// TwinCAT 3 PLC project Depal2
// libraries:
//   Tc2_Standard, * (Beckhoff Automation GmbH)
//   Tc2_System, * (Beckhoff Automation GmbH)
//   Tc3_Module, * (Beckhoff Automation GmbH)
// project tree:
//   Global Variables/ Global_Variables.TcGVL, Global_Variables_HMI.TcGVL, Global_Variables_sBool.TcGVL, Variable_Configuration.TcGVL
//   POUs/Function Blocks/ TOGGLE.TcPOU
//   POUs/ IOLink.TcPOU, MAIN.TcPOU, Messages.TcPOU, Tiersheet_Car.TcPOU
//   / Standard.TcTTO
// real-time tasks:
//   TASK Standard: cycle T#10ms, priority 20, ADS port 350
// I/O:
//   DEVICE Depal 2 I/O, AmsNetId 5.155.243.167.3.1
//     Term 1 (EK1200) [EK1200-5000 EtherCAT Power supply (2A E-Bus)]
//       Term 2 (EK1122) [EK1122 2 port EtherCAT junction]
//         IO-Link1 (ifm IO-Link Master AL1332) [ifm IO-Link Master AL1332]
//           modules: Module 1 (IOL_In_8Byte), Module 2 (IOL_In_8Byte), Module 3 (IOL_In_8Byte), Module 4 (IOL_In_8Byte), Module 5 (IOL_In_8Byte), Module 6 (IOL_In_8Byte), Module 7 (IOL_In_8Byte), Module 8 (IOL_In_8Byte)
//         IO-Link2 (ifm IO-Link Master AL1332) [ifm IO-Link Master AL1332]
//           modules: Module 1 (IOL_In_8Byte), Module 2 (IOL_In_8Byte), Module 3 (IOL_In_8Byte), Module 4 (IOL_In_8Byte), Module 5 (IOL_In_8Byte), Module 6 (IOL_In_8Byte), Module 7 (IOL_In_8Byte), Module 8 (IOL_In_8Byte)
//         IO-Link3 (ifm IO-Link Master AL1332) [ifm IO-Link Master AL1332]
//           modules: Module 1 (IOL_In_8Byte), Module 2 (IOL_In_8Byte), Module 3 (IOL_In_8Byte), Module 4 (IOL_In_8Byte), Module 5 (IOL_In_8Byte), Module 6 (IOL_In_8Byte), Module 7 (IOL_In_8Byte), Module 8 (IOL_In_8Byte)
//         IO-Link4 (ifm IO-Link Master AL1332) [ifm IO-Link Master AL1332]
//           modules: Module 1 (IOL_In_8Byte), Module 2 (IOL_In_8Byte), Module 3 (IOL_In_8Byte), Module 4 (IOL_In_8Byte), Module 5 (IOL_In_8Byte), Module 6 (IOL_In_8Byte), Module 7 (IOL_In_8Byte), Module 8 (IOL_In_8Byte)
//         IO-Link5 (ifm IO-Link Master AL1332) [ifm IO-Link Master AL1332]
//           modules: Module 1 (IOL_In_8Byte), Module 2 (Digital_IN), Module 3 (Digital_IN), Module 4 (IOL_In_8Byte), Module 5 (IOL_In_8Byte), Module 6 (IOL_In_8Byte), Module 7 (IOL_In_8Byte), Module 8 (IOL_In_8Byte)
//       Box 4 (BK1250)
// variable links:
//   Depal2/Depal2 Instance <-> Depal 2 I/O/Term 1 (EK1200)/Box 4 (BK1250)
//     Standard Inputs/.i453 <-> Term 7 (KL1114)/Channel 4/Input
//     Standard Inputs/.iCarriage_VAC <-> Term 2 (KL1114)/Channel 3/Input
//     Standard Inputs/.iCarriage_Vfd <-> Term 5 (KL1114)/Channel 3/Input
//     Standard Inputs/.iChain_Hoist_VAC <-> Term 2 (KL1114)/Channel 2/Input
//     Standard Inputs/.iChain_Hoist_Vfd <-> Term 5 (KL1114)/Channel 2/Input
//     Standard Inputs/.iChamber_Chain_VAC <-> Term 2 (KL1114)/Channel 4/Input
//     Standard Inputs/.iChamber_Chain_Vfd <-> Term 5 (KL1114)/Channel 4/Input
//     Standard Inputs/.iDM2_EmergencyStop <-> Term 8 (KL9260)/Channel 1/Power
//     Standard Inputs/.iDM2_Fuse <-> Term 8 (KL9260)/Channel 1/ShortCircuit
//     Standard Inputs/.iDischarge1_VAC <-> Term 4 (KL1114)/Channel 1/Input
//     Standard Inputs/.iDischarge2_VAC <-> Term 4 (KL1114)/Channel 2/Input
//     Standard Inputs/.iDischarge3_VAC <-> Term 4 (KL1114)/Channel 3/Input
//     Standard Inputs/.iDischarge1_Vfd <-> Term 7 (KL1114)/Channel 1/Input
//     Standard Inputs/.iDischarge2_Vfd <-> Term 7 (KL1114)/Channel 2/Input
//     Standard Inputs/.iDischarge3_Vfd <-> Term 7 (KL1114)/Channel 3/Input
//     Standard Inputs/.iPallet_Discharge_VAC <-> Term 3 (KL1114)/Channel 1/Input
//     Standard Inputs/.iPallet_Discharge_Vfd <-> Term 6 (KL1114)/Channel 1/Input
//     Standard Inputs/.iPallet_Infeed1_VAC <-> Term 3 (KL1114)/Channel 2/Input
//     Standard Inputs/.iPallet_Infeed2_VAC <-> Term 3 (KL1114)/Channel 3/Input
//     Standard Inputs/.iPallet_Infeed1_Vfd <-> Term 6 (KL1114)/Channel 2/Input
//     Standard Inputs/.iPallet_Infeed2_Vfd <-> Term 6 (KL1114)/Channel 3/Input
//     Standard Inputs/.iProductHeight_SweepPos <-> Term 4 (KL1114)/Channel 4/Input
//     Standard Inputs/.iTable_Top_VAC <-> Term 2 (KL1114)/Channel 1/Input
//     Standard Inputs/.iTable_Top_Vfd <-> Term 5 (KL1114)/Channel 1/Input
//     Standard Inputs/.iTierSheet_Car_VAC <-> Term 3 (KL1114)/Channel 4/Input
//     Standard Inputs/.iTierSheet_Car_Vfd <-> Term 6 (KL1114)/Channel 4/Input
//     Standard Outputs/.oBrake_Carriage <-> Term 30 (KL2612)/Channel 2/Output
//     Standard Outputs/.oBrake_Hoist <-> Term 30 (KL2612)/Channel 1/Output
//     Standard Outputs/.oCarriage_Forward <-> Term 25 (KL2612)/Channel 1/Output
//     Standard Outputs/.oCarriage_Reverse <-> Term 25 (KL2612)/Channel 2/Output
//     Standard Outputs/.oCarriage_Slow <-> Term 21 (KL2612)/Channel 2/Output
//     Standard Outputs/.oChainHoist_Down <-> Term 24 (KL2612)/Channel 2/Output
//     Standard Outputs/.oChainHoist_Up <-> Term 24 (KL2612)/Channel 1/Output
//     Standard Outputs/.oChainHoist_Up_Slow <-> Term 32 (KL2612)/Channel 1/Output
//     Standard Outputs/.oChainberChainRev <-> Term 32 (KL2612)/Channel 2/Output
//     Standard Outputs/.oDischarge1_Run <-> Term 28 (KL2612)/Channel 2/Output
//     Standard Outputs/.oDischarge2_Run <-> Term 29 (KL2612)/Channel 1/Output
//     Standard Outputs/.oElevator_Infeed <-> Term 26 (KL2612)/Channel 1/Output
//     Standard Outputs/.oHoistDoors_Close <-> Term 13 (KL2612)/Channel 2/Output
//     Standard Outputs/.oHoistDoors_Open <-> Term 13 (KL2612)/Channel 1/Output
//     Standard Outputs/.oHoist_Shrouds_Close <-> Term 12 (KL2612)/Channel 1/Output
//     Standard Outputs/.oHoist_Shrouds_Open <-> Term 12 (KL2612)/Channel 2/Output
//     Standard Outputs/.oIndicator_Green <-> Term 22 (KL2612)/Channel 1/Output
//     Standard Outputs/.oIndicator_Red <-> Term 23 (KL2612)/Channel 1/Output
//     Standard Outputs/.oIndicator_Yellow <-> Term 22 (KL2612)/Channel 2/Output
//     Standard Outputs/.oInfeed1Rev <-> Term 29 (KL2612)/Channel 2/Output
//     Standard Outputs/.oInfeed2Rev <-> Term 33 (KL2612)/Channel 1/Output
//     Standard Outputs/.oLayer_Capture <-> Term 14 (KL2612)/Channel 1/Output
//     Standard Outputs/.oLayer_Release <-> Term 14 (KL2612)/Channel 2/Output
//     Standard Outputs/.oPalletDischarge_Run <-> Term 26 (KL2612)/Channel 2/Output
//     Standard Outputs/.oPalletInfeed1_Run <-> Term 27 (KL2612)/Channel 1/Output
//     Standard Outputs/.oPalletInfeed2_Run <-> Term 27 (KL2612)/Channel 2/Output
//     Standard Outputs/.oSweepGate_Close <-> Term 9 (KL2612)/Channel 2/Output
//     Standard Outputs/.oSweepGate_Open <-> Term 9 (KL2612)/Channel 1/Output
//     Standard Outputs/.oSweepgate_Engage <-> Term 15 (KL2612)/Channel 1/Output
//     Standard Outputs/.oSweepgate_Release <-> Term 15 (KL2612)/Channel 2/Output
//     Standard Outputs/.oTableTop_Run <-> Term 23 (KL2612)/Channel 2/Output
//     Standard Outputs/.oTierSheetGripper_Engage <-> Term 16 (KL2612)/Channel 1/Output
//     Standard Outputs/.oTierSheetGripper_Release <-> Term 16 (KL2612)/Channel 2/Output
//     Standard Outputs/.oTierSheet_Bin_Close <-> Term 17 (KL2612)/Channel 2/Output
//     Standard Outputs/.oTierSheet_Bin_Open <-> Term 17 (KL2612)/Channel 1/Output
//     Standard Outputs/.oTierSheet_Car_Brake <-> Term 28 (KL2612)/Channel 1/Output
//     Standard Outputs/.oTierSheet_Car_Fwd <-> Term 31 (KL2612)/Channel 1/Output
//     Standard Outputs/.oTierSheet_Car_Rev <-> Term 31 (KL2612)/Channel 2/Output
//     Standard Outputs/.oTiersheetRemover_Down <-> Term 10 (KL2612)/Channel 2/Output
//     Standard Outputs/.oTiersheetRemover_Up <-> Term 10 (KL2612)/Channel 1/Output
//     Standard Outputs/.oTopFrame_Bin_Close <-> Term 18 (KL2612)/Channel 2/Output
//     Standard Outputs/.oTopFrame_Bin_Open <-> Term 18 (KL2612)/Channel 1/Output
//     Standard Outputs/.oTopFrame_Remover_Clamps_Engage <-> Term 20 (KL2612)/Channel 1/Output
//     Standard Outputs/.oTopFrame_Remover_Clamps_Release <-> Term 20 (KL2612)/Channel 2/Output
//     Standard Outputs/.oTopFrame_Remover_Lock <-> Term 19 (KL2612)/Channel 1/Output
//     Standard Outputs/.oTopFrame_Remover_Unlock <-> Term 19 (KL2612)/Channel 2/Output
//     Standard Outputs/.oTopFrame_Seize <-> Term 11 (KL2612)/Channel 2/Output
//     Standard Outputs/.oTrolleySlowdown <-> Term 33 (KL2612)/Channel 2/Output
//     Standard Outputs/.oVacuum_Engage <-> Term 21 (KL2612)/Channel 1/Output
//     Standard Outputs/.oVacuum_Solenoid <-> Term 11 (KL2612)/Channel 1/Output
//   Depal2/Depal2 Instance <-> Depal 2 I/O/Term 1 (EK1200)/Term 2 (EK1122)/IO-Link1 (ifm IO-Link Master AL1332)
//     Standard Inputs/.i1X01_HoistDoors_Closed <-> Module 1 (IOL_In_8Byte)/TxPDO/input byte 0
//     Standard Inputs/.i1X02_HoistLiftDown_Slowdown <-> Module 2 (IOL_In_8Byte)/TxPDO/input byte 0
//     Standard Inputs/.i1X03_HoistLift_Down <-> Module 3 (IOL_In_8Byte)/TxPDO/input byte 0
//     Standard Inputs/.i1X04_Hoist_Discharge_Jam <-> Module 4 (IOL_In_8Byte)/TxPDO/input byte 0
//     Standard Inputs/.i1X05_Infeed1_Pallet <-> Module 5 (IOL_In_8Byte)/TxPDO/input byte 0
//     Standard Inputs/.i1X06_Infeed2_Pallet <-> Module 6 (IOL_In_8Byte)/TxPDO/input byte 0
//     Standard Inputs/.i1X07_Pallet_in_Hoist <-> Module 7 (IOL_In_8Byte)/TxPDO/input byte 0
//     Standard Inputs/.i1X08_1114 <-> Module 8 (IOL_In_8Byte)/TxPDO/input byte 0
//   Depal2/Depal2 Instance <-> Depal 2 I/O/Term 1 (EK1200)/Term 2 (EK1122)/IO-Link2 (ifm IO-Link Master AL1332)
//     Standard Inputs/.i2X01 <-> Module 1 (IOL_In_8Byte)/TxPDO/input byte 0
//     Standard Inputs/.i2X02_HoistLift_Up <-> Module 2 (IOL_In_8Byte)/TxPDO/input byte 0
//     Standard Inputs/.i2X03_HoistLift_LastTier <-> Module 3 (IOL_In_8Byte)/TxPDO/input byte 0
//     Standard Inputs/.i2X04_Top_Frame_Monitor <-> Module 4 (IOL_In_8Byte)/TxPDO/input byte 0
//     Standard Inputs/.i2X05_DunnageBin_Full <-> Module 5 (IOL_In_8Byte)/TxPDO/input byte 0
//     Standard Inputs/.i2X06_TableTop_Accumulation <-> Module 6 (IOL_In_8Byte)/TxPDO/input byte 0
//     Standard Inputs/.i2X07_SingleFiler_Accumulation <-> Module 7 (IOL_In_8Byte)/TxPDO/input byte 0
//     Standard Inputs/.i2X08_CanTrack_Accumulation <-> Module 8 (IOL_In_8Byte)/TxPDO/input byte 0
//   Depal2/Depal2 Instance <-> Depal 2 I/O/Term 1 (EK1200)/Term 2 (EK1122)/IO-Link3 (ifm IO-Link Master AL1332)
//     Standard Inputs/.i3X01_SweepGateDoor_Open <-> Module 1 (IOL_In_8Byte)/TxPDO/input byte 0
//     Standard Inputs/.i3X02_CarriageRetract_Slowdown <-> Module 2 (IOL_In_8Byte)/TxPDO/input byte 0
//     Standard Inputs/.i3X03_Carriage_Retracted <-> Module 3 (IOL_In_8Byte)/TxPDO/input byte 0
//     Standard Inputs/.i3X04_Carriage_Extended <-> Module 4 (IOL_In_8Byte)/TxPDO/input byte 0
//     Standard Inputs/.i3X05_CarriageExtend_Slowdown <-> Module 5 (IOL_In_8Byte)/TxPDO/input byte 0
//     Standard Inputs/.i3X06_Layer_Capture_Monitor <-> Module 6 (IOL_In_8Byte)/TxPDO/input byte 0
//     Standard Inputs/.i3X07_Vacuum_On <-> Module 7 (IOL_In_8Byte)/TxPDO/input byte 0
//     Standard Inputs/.i3X08_ <-> Module 8 (IOL_In_8Byte)/TxPDO/input byte 0
//   Depal2/Depal2 Instance <-> Depal 2 I/O/Term 1 (EK1200)/Term 2 (EK1122)/IO-Link4 (ifm IO-Link Master AL1332)
//     Standard Inputs/.i4X01_Trolley_at_Hoist <-> Module 1 (IOL_In_8Byte)/TxPDO/input byte 0
//     Standard Inputs/.i4X02_Trolley_at_Hoist_Slowdown <-> Module 2 (IOL_In_8Byte)/TxPDO/input byte 0
//     Standard Inputs/.i4X03_Trolley_at_TierSheet_Bin_Slowdown <-> Module 3 (IOL_In_8Byte)/TxPDO/input byte 0
//     Standard Inputs/.i4X04_Trolley_at_TierSheetBin <-> Module 4 (IOL_In_8Byte)/TxPDO/input byte 0
//     Standard Inputs/.i4X05_Trolley_at_TopframeBin_Slowdown <-> Module 5 (IOL_In_8Byte)/TxPDO/input byte 0
//     Standard Inputs/.i4X06_Trolley_at_TopframeBin <-> Module 6 (IOL_In_8Byte)/TxPDO/input byte 0
//     Standard Inputs/.i4X07_TierSheetBin_Full <-> Module 7 (IOL_In_8Byte)/TxPDO/input byte 0
//     Standard Inputs/.i4X08_TopframeBin_Full <-> Module 8 (IOL_In_8Byte)/TxPDO/input byte 0
//   Depal2/Depal2 Instance <-> Depal 2 I/O/Term 1 (EK1200)/Term 2 (EK1122)/IO-Link5 (ifm IO-Link Master AL1332)
//     Standard Inputs/.i5X01_TierSheet_Vacuum_Monitor <-> Module 1 (IOL_In_8Byte)/TxPDO/input byte 0
//     Standard Inputs/.i5X02_TierSheet_Remover_Down <-> Module 2 (Digital_IN)/TxPDO/input byte 0
//     Standard Inputs/.i5X03_TiersheetRemoverUp <-> Module 3 (Digital_IN)/TxPDO/input byte 0
//     Standard Inputs/.i5X04_ <-> Module 4 (IOL_In_8Byte)/TxPDO/input byte 0
//     Standard Inputs/.i5X08_ <-> Module 8 (IOL_In_8Byte)/TxPDO/input byte 0
//     Standard Inputs/.i5X05_Topframe_Remover_Up <-> Module 5 (IOL_In_8Byte)/TxPDO/input byte 0
//     Standard Inputs/.i5X06_Topframe_On_BoardA <-> Module 6 (IOL_In_8Byte)/TxPDO/input byte 0
//     Standard Inputs/.i5X07_Topframe_On_BoardB <-> Module 7 (IOL_In_8Byte)/TxPDO/input byte 0

CONFIGURATION Depal2
    RESOURCE PLC ON TwinCAT3
        TASK Standard(INTERVAL := T#10ms, PRIORITY := 20);
        PROGRAM MAIN WITH Standard : MAIN;
    END_RESOURCE
END_CONFIGURATION

// ---- Global Variables/Global_Variables.TcGVL
{attribute 'Tc2GvlVarNames'}
VAR_GLOBAL
(***********************IO-LINK  INPUT************************************)
(**IO-Link1 AL1332**)
	i1X01_HoistDoors_Closed AT %I*:USINT;
	i1X02_HoistLiftDown_Slowdown AT %I*:USINT;
	i1X03_HoistLift_Down AT %I*:USINT;
	i1X04_Hoist_Discharge_Jam AT %I*:USINT;
	i1X05_Infeed1_Pallet AT %I*:USINT;
	i1X06_Infeed2_Pallet  AT %I*:USINT;
	i1X07_Pallet_in_Hoist AT %I*:USINT;
	i1X08_1114 AT %I*:USINT;

(**IO-Link2 AL1332**)
	i2X01 AT %I*:USINT;
	i2X02_HoistLift_Up AT %I*:USINT;
	i2X03_HoistLift_LastTier  AT %I*:USINT;
	i2X04_Top_Frame_Monitor AT %I*:USINT;
	i2X05_DunnageBin_Full AT %I*:USINT;
	i2X06_TableTop_Accumulation  AT %I*:USINT;
	i2X07_SingleFiler_Accumulation  AT %I*:USINT;
	i2X08_CanTrack_Accumulation  AT %I*:USINT;

(**IO-Link3 AL1332**)
	i3X01_SweepGateDoor_Open AT %I*:USINT;
	i3X02_CarriageRetract_Slowdown AT %I*:USINT;
	i3X03_Carriage_Retracted AT %I*:USINT;
	i3X04_Carriage_Extended AT %I*:USINT;
	i3X05_CarriageExtend_Slowdown AT %I*:USINT;
	i3X06_Layer_Capture_Monitor AT %I*:USINT;
	i3X07_Vacuum_On AT %I*:USINT;
	i3X08_ AT %I*:USINT;

(**IO-Link4 AL1332**)
	i4X01_Trolley_at_Hoist AT %I*:USINT;
	i4X02_Trolley_at_Hoist_Slowdown AT %I*:USINT;
	i4X03_Trolley_at_TierSheet_Bin_Slowdown AT %I*:USINT;
	i4X04_Trolley_at_TierSheetBin AT %I*:USINT;
	i4X05_Trolley_at_TopframeBin_Slowdown AT %I*:USINT;
	i4X06_Trolley_at_TopframeBin AT %I*:USINT;
	i4X07_TierSheetBin_Full AT %I*:USINT;
	i4X08_TopframeBin_Full AT %I*:USINT;

(**IO-Link5 AL1332**)
	i5X01_TierSheet_Vacuum_Monitor AT %I*:USINT;
	i5X02_TierSheet_Remover_Down AT %I*:USINT;
	i5X03_TiersheetRemoverUp AT %I*:USINT;
	i5X04_ AT %I*:USINT;
	i5X05_Topframe_Remover_Up AT %I*:USINT;
	i5X06_Topframe_On_BoardA AT %I*:USINT;
	i5X07_Topframe_On_BoardB AT %I*:USINT;
	i5X08_ AT %I*:USINT;

(**Slot 2 KL-1114*)(*VAC Disconnect*)
	iTable_Top_VAC AT %I*:BOOL;
	iChain_Hoist_VAC AT %I*:BOOL;
	iCarriage_VAC AT %I*:BOOL;
	iChamber_Chain_VAC AT %I*:BOOL;

(**Slot 3 KL1114*)(*VAC Disconnect*)
	iPallet_Discharge_VAC AT %I*:BOOL;
	iPallet_Infeed1_VAC AT %I*:BOOL;
	iPallet_Infeed2_VAC AT %I*:BOOL;
	iTierSheet_Car_VAC AT %I*:BOOL;

(**Slot 4 KL1114*)(*VAC Disconnect*)
	iDischarge1_VAC AT %I*:BOOL;
	iDischarge2_VAC AT %I*:BOOL;
	iDischarge3_VAC AT %I*:BOOL;
	iProductHeight_SweepPos AT %I*:BOOL;
	
(**Slot 5 KL1114*)(*VFD ENABLE*)
	iTable_Top_Vfd AT %I*:BOOL;
	iChain_Hoist_Vfd AT %I*:BOOL;
	iCarriage_Vfd AT %I*:BOOL;
	iChamber_Chain_Vfd AT %I*:BOOL;

(**Slot 6 KL1114*)(*VFD ENABLE*)
	iPallet_Discharge_Vfd AT %I*:BOOL;
	iPallet_Infeed1_Vfd AT %I*:BOOL;
	iPallet_Infeed2_Vfd AT %I*:BOOL;
	iTierSheet_Car_Vfd AT %I*:BOOL;

(**Slot 7 KL1114*)(*VFD ENABLE*)
	iDischarge1_Vfd AT %I*:BOOL;
	iDischarge2_Vfd AT %I*:BOOL;
	iDischarge3_Vfd AT %I*:BOOL;
	i453 AT %I*:BOOL;

(** Slot 8 KL-9260*)
	iDM2_EmergencyStop AT %I*:BOOL;
	iDM2_Fuse AT %I*:BOOL;
(**Slot 9 KL-2602*)
	oSweepGate_Open AT %Q*:BOOL;
	oSweepGate_Close AT %Q*:BOOL;

(**Slot 10 KL-2602*)
	oTiersheetRemover_Up AT %Q*:BOOL;
	oTiersheetRemover_Down AT %Q*:BOOL;

(**Slot 11 KL-2602*)
	oVacuum_Solenoid AT %Q*:BOOL;
	oTopFrame_Seize AT %Q*:BOOL;

(**Slot 12 KL-2602*)
	oHoist_Shrouds_Close AT %Q*:BOOL;
	oHoist_Shrouds_Open AT %Q*:BOOL;

(**Slot 13 KL-2602*)
	oHoistDoors_Open AT %Q*:BOOL;
	oHoistDoors_Close AT %Q*:BOOL;

(**Slot 14 KL-2602*)
	oLayer_Capture AT %Q*:BOOL;
	oLayer_Release AT %Q*:BOOL;
(**Slot 15 KL-2602*)
	oSweepgate_Engage AT %Q*:BOOL;
	oSweepgate_Release AT %Q*:BOOL;

(**Slot 16 KL-2602*)
	oTierSheetGripper_Engage AT %Q*:BOOL;
	oTierSheetGripper_Release AT %Q*:BOOL;

(**Slot 17 KL-2602*)
	oTierSheet_Bin_Open AT %Q*:BOOL;
	oTierSheet_Bin_Close AT %Q*:BOOL;

(**Slot 18 KL-2602*)
	oTopFrame_Bin_Open AT %Q*:BOOL;
	oTopFrame_Bin_Close AT %Q*:BOOL;

(**Slot 19 KL-2602*)
	oTopFrame_Remover_Lock AT %Q*:BOOL;
	oTopFrame_Remover_Unlock AT %Q*:BOOL;

(**Slot 20 KL-2602*)
	oTopFrame_Remover_Clamps_Engage AT %Q*:BOOL;
	oTopFrame_Remover_Clamps_Release AT %Q*:BOOL;

(**Slot 21 KL-2602*)
	oVacuum_Engage AT %Q*:BOOL;
	oCarriage_Slow AT %Q*:BOOL;

(**Slot 22 KL-2612*)
	oIndicator_Green AT %Q*:BOOL;
	oIndicator_Yellow AT %Q*:BOOL;

(*Slot 23 KL-2612*)
	oIndicator_Red AT %Q*:BOOL;
	oTableTop_Run AT %Q*:BOOL;

(*Slot 24 KL-2612*)
	oChainHoist_Up AT %Q*:BOOL;
	oChainHoist_Down AT %Q*:BOOL;

(*Slot 25 KL-2612*)
	oCarriage_Forward AT %Q*:BOOL;
	oCarriage_Reverse AT %Q*:BOOL;

(*Slot 26 KL-2612*)
	oElevator_Infeed AT %Q*:BOOL;
	oPalletDischarge_Run AT %Q*:BOOL;

(*Slot 27 KL-2612*)
	oPalletInfeed1_Run AT %Q*:BOOL;
	oPalletInfeed2_Run AT %Q*:BOOL;
(*Slot 28 KL-2612*)
	oTierSheet_Car_Brake AT %Q*:BOOL;
	oDischarge1_Run AT %Q*:BOOL;

(*Slot 29 KL-2612*)
	oDischarge2_Run AT %Q*:BOOL;
	oInfeed1Rev AT %Q*:BOOL;

(*Slot 30 KL-2612*)
	oBrake_Hoist AT %Q*:BOOL;
	oBrake_Carriage AT %Q*:BOOL;

(*Slot 31 KL-2612*)
	oTierSheet_Car_Fwd AT %Q*:BOOL;
	oTierSheet_Car_Rev AT %Q*:BOOL;

(*Slot 32 KL-2612*)
	oChainHoist_Up_Slow AT %Q*:BOOL;
	oChainberChainRev AT %Q*:BOOL;

(*Slot 33 KL-2612*)
	oInfeed2Rev AT %Q*:BOOL;
	oTrolleySlowdown AT %Q*:BOOL;

(***********IOLink Int to Bool*********)


	Infeed2_Pallet: BOOL;
	Infeed1_Pallet: BOOL;

	Pallet_in_Hoist: BOOL;
	Hoist_Discharge_Jam: BOOL;

	HoistDoors_Closed: BOOL;

	CanTrack_Accumulation: BOOL;
	SingleFiler_Accumulation: BOOL;
	TableTop_Accumulation: BOOL;

	DunnageBin_Full: BOOL;
	Top_Frame_Monitor: BOOL;
	HoistLift_LastTier: BOOL;
	HoistLiftDown_Slowdown: BOOL;

	HoistLift_Up: BOOL;
	HoistLift_Down: BOOL;

	SweepGateDoor_Open: BOOL;

	CarriageRetract_Slowdown: BOOL;
	Carriage_Retracted: BOOL;
	Carriage_Extended: BOOL;
	CarriageExtend_Slowdown: BOOL;


	Vacuum_On: BOOL;

	Trolley_at_Hoist: BOOL;
	Trolley_at_Hoist_Slowdown: BOOL;

	Trolley_at_TierSheet_Bin_Slowdown: BOOL;
	Trolley_at_TierSheetBin: BOOL;

	Trolley_at_TopframeBin_Slowdown: BOOL;
	Trolley_at_TopframeBin: BOOL;

	TierSheetBin_Full: BOOL;
	TopframeBin_Full: BOOL;

	TierSheet_Vacuum_Monitor: BOOL;

	TierSheet_Trolley_at_Hoist_Slowdown: BOOL;
	TierSheet_Trolley_at_TierSheet_Bin_Slowdown: BOOL;

	Topframe_Remover_Up: BOOL;
	Topframe_On_BoardA: BOOL;
	Topframe_On_BoardB: BOOL;












	M2CanCounter: CTU;
	LINC: BOOL;
	sc_Depal2Count: INT;
	sc_Depal2_1stShift: BOOL;
	sc_Depal2_1stShiftStart: BOOL;
	sc_M1CC1stReset: BOOL;
	_1stshiftcnt: CTU;
	jsjs: CTU;
	sc_Depal2_2NDShiftStart: BOOL;
	Pallet_Counter: CTU;
	HoistDoorsOpen: BOOL;
END_VAR

// ---- Global Variables/Global_Variables_HMI.TcGVL
{attribute 'Tc2GvlVarNames'}
VAR_GLOBAL
	sEmergencyStop:BOOL;
	EmergencyStop_Latch:BOOL;
	sEstop_Reset:BOOL;
	sMessages: STRING;
	CC2_Count: REAL;
	CC2_Reset:BOOL;
	sManual: BOOL;
	sManualLt: BOOL;
	sElevator_Infeed: BOOL;
	sHoist_UP: BOOL;
	sHoist_DN: BOOL;
	sCar_Fwd: BOOL;
	sCar_Rev: BOOL;
	sGateOpen: BOOL;
	sTableTop: BOOL;
	sDischarge1: BOOL;
	sDischarge2: BOOL;
	sDischarge3: BOOL;
	sTrCar_Fwd: BOOL;
	sTrCar_Rev: BOOL;
	Auto: BOOL;
	sAuto: BOOL;
	sAutoLt:BOOL;
	Manual: BOOL;
	sManualLoading: BOOL;
	Manual_Loading: BOOL;
	sAutoLoading: BOOL;
	sManualLoadingLt: BOOL;
	sAutoLoadingLt: BOOL;
	Auto_Loading: BOOL;
	sReset: BOOL;
	sInfeed1Rev: BOOL;
	sInfeed2Rev: BOOL;
	sElevator_Conv_Rev: BOOL;
	sInfeed2: BOOL;
	sInfeed1: BOOL;
	sNew_PalletLt: BOOL;
	Stop_For_Frame_Remove: BOOL;
	sStop_For_Frame_RemoveLt: BOOL;
	sc_Depal2_1stshiftcount: INT;
	sc_Depal2_2NDshiftcount: INT;
	sStopHoist: BOOL;
	StopHoistLt: BOOL;
	TrolleyEnable: BOOL;
	Remover_Oneshot: TP;
	TierSheet_Remover_Down:BOOL;
	sTopFrame_RemovalLt: BOOL;
	sTopFrame_Removal: BOOL;
	sTrolleyAuto: BOOL;
	sTrolleyAutoLt: BOOL;

	sTrolleytoFrameBin: BOOL;
	sTrolleytoHoist: BOOL;
	sTrolleytoSheetBin: BOOL;
	sTierSheetRemover_UpLT: BOOL;

	Transfer_Can_to_Table: BOOL;
	Carriage_to_Table: BOOL;
	sTop_Frame_Removed: BOOL;
	sTableTopLt: BOOL;
	sDisch1Lt: BOOL;
	sDisch2Lt: BOOL;
	sDisch1FullLt: BOOL;
	sDisch2FullLt: BOOL;
	sDischargeTT_FullLt: BOOL;

	sFrameClamps: BOOL;
	sVac: BOOL;
	sTiersheetRemover_Down: BOOL;
	SheetRemoverToggle: TOGGLE;
	sTiersheetRemover_Up: BOOL;
	sHoistLT: BOOL;
	sToHoistLT: BOOL;
	sSheetBinLT: BOOL;
	sToSheetBinLT: BOOL;
	sToFrameBinLT: BOOL;
	sFrameBinLT: BOOL;
	sFrame_Remover: BOOL;

	s1: BOOL;
	s2: BOOL;
	s3: BOOL;
	s4: BOOL;
	s5: BOOL;
	s6: BOOL;
	s7: BOOL;
	s8: BOOL;
	s9: BOOL;
	s10: BOOL;
	s11: BOOL;
	s12: BOOL;
	s13: BOOL;
	s14: BOOL;
	s15: BOOL;
	s16: BOOL;
	s17: BOOL;
	s18: BOOL;
	s19: BOOL;
	s20: BOOL;

	s21: BOOL;
	s22: BOOL;

	s23: BOOL;
	s24: BOOL;

	s25: BOOL;
	s26: BOOL;

	s27: BOOL;
	s28: BOOL;

	s29: BOOL;
	s30: BOOL;

	s31: BOOL;
	s32: BOOL;


	sMsg1: STRING;
	sMsg2: STRING;
	sMsg3: STRING;
	sMsg4: STRING;
	sMsg5: STRING;
	sMsg6: STRING;
	sMsg7: STRING;
	sMsg8: STRING;
	sMsg9: STRING;
	sMsg10: STRING;
	sMsg11: STRING;
	sMsg12: STRING;
	sMsg13: STRING;
	sMsg14: STRING;
	sMsg15: STRING;
	sMsg16: STRING;
	sMsg17: STRING;
	sMsg18: STRING;
	sMsg19: STRING;
	sMsg20: STRING;
	scM2CanReset: BOOL;
	scM2CanCount: REAL;
	scDepal_2_CanCountReset: BOOL;
	scDepal_2_CanCount: REAL;
END_VAR

// ---- Global Variables/Global_Variables_sBool.TcGVL
{attribute 'Tc2GvlVarNames'}
VAR_GLOBAL
	sCan_Discharge_Enable:BOOL;
	Pallet_Jam_Alarm: BOOL;
	Last_Can_Tier:BOOL;
	sNew_Pallet: BOOL;
	TiersheetRemover_Up:BOOL;

	Trolley_Disable: BOOL;
	Layer_Capture_Monitor: BOOL;

END_VAR

// ---- Global Variables/Variable_Configuration.TcGVL
{attribute 'Tc2GvlVarNames'}
VAR_CONFIG
END_VAR

// ---- POUs/MAIN.TcPOU

PROGRAM MAIN
VAR



	SGO: TOGGLE;
	SGC: TOGGLE;
	TRU: TOGGLE;
	TRD: TOGGLE;
	VS: TOGGLE;
	TFS: TOGGLE;
	HSC: TOGGLE;
	HSO: TOGGLE;
	HDO: TOGGLE;
	HDC: TOGGLE;
	LC: TOGGLE;
	LR: TOGGLE;


	Eject_Empty_Pallet: BOOL;
	Empty_Pallet_Ejecting: BOOL;
	Empty_Pallet: BOOL;
	Full_Pallet: BOOL;
	Shroud_Latch: BOOL;


	Hoist_Cycle: BOOL;
	Next_Tier: BOOL;
	Hoist_Up_Disable: BOOL;
	ChainHoist_Enable: BOOL;
	Rev_Enable: BOOL;

	Auto_Tog: TOGGLE;



	Delay_Pallet_Advance2: TON;

	Delay_Pallet_Advance: TON;
	sChamberChain_Run: BOOL;
	Hoist_Down_Complete_TMR: TON;
	Discharge1_Pallet: BOOL;
	Eject_Cycle_TMR: TON;
	Hoist_Up_Tog: TOGGLE;
	Height_TMR: TOF;
	Reset_One_Shot: TP;
	sHoistUpDisable: BOOL;
	sChainHoistDn: BOOL;
	Fwd_Delay: TON;
	sCarriage_to_Pickup: BOOL;

	Open_Delay: TON;

	Release_Capture: TOF;
	DR2_Tog: TOGGLE;
	DR3_Tog: TOGGLE;
	DR4_Tog: TOGGLE;
	HoistUpDisableTog: TOGGLE;
	Gate_Closure_TMR:TON;




	Pa1Tog: TOGGLE;
	OpenTMR: TOF;
	CloseTMR: TOF;
	Down_Slow_Delay: TON;
	DSD: TIME;
	test: BOOL;
	Last_TierTMR1: TOF;
	Last_TierTMR2: TON;

	Down_Completion_TMR: TOF;
	Maintainloading: TOF;
	Ejecting_Pallet: BOOL;
	EmptyPallet_Jam_TMR: TON;





	TopFrameRem: TOF;
	Hoist_OneShot: TP;
	Hoist_Dn_Fast_Limit: TON;
	HDFL: TIME;
	Carriage_Disable_For_New_Pallet: BOOL;
	Slow_Reset: TP;
	LCT_Maintain: TOF;
	TT_Maintain: TOF;
	Disch1_Maintain: TOF;
	Disch2_Maintain: TOF;



	AutoLoadingTog: TOGGLE;
	ManualLoadingTog: TOGGLE;

	StopHoist_Tog: TOGGLE;

	TableTopJam: TON;
	Disch2Delay: TON;

	Discharge2Jam: TON;


	Disch2Full: TON;
	DR3TP: TP;
	Discharge2TOG: TOGGLE;
	Can_Count_M2: CTU;
	CC2: REAL;
	CanCount2A: CTU;
	CanCount2B: CTU;
	CC2B: REAL;
	CanCntReset: BOOL;
	CC2_Tens: REAL;

	FwdMaintain: TOF;
	Top_Frame_Removal: TON;
	Carriage_Forward_Enable: BOOL;
	Close_Pulse: TP;
	TT_Jam_Manager: TOF;
	Reverse_Delay: TON;
	Flash1_NP: TON;
	Flash2_NP: TOF;


	Flash1B: TON;
	Flash2B: TOF;
	mt: TOF;
	SlowTest: BOOL;
	Down_Slow_Maintain: TOF;
	Last_Slip_Sheet: TON;
	Test1: BOOL;
	Test2: BOOL;
	Empty_Pallet_Pulse: TP;
	Clank2_TMR: TON;
	Discharge_Run_TMR: TOF;
	Carriage_Slow_Enable: BOOL;
	Slow_Maintain: TOF;
	sc_DepalM2Count: INT;
	M2CanCounter2: CTU;
	M2CanCounter3: CTU;
	sc_Depal2Count3: BOOL;
	sc_Depal2Count2: BOOL;
	sc_Depal2Count13: INT;
	sc_Depal2Count12: INT;
	M2CanCounter4: CTU;
	M2CanCounter33: CTU;
	M2CanCounter34: CTU;
	a: INT;
	b: INT;
	C: INT;
	M2CanCounter333: CTU;
	d: INT;
	e: INT;
	F: INT;
	M2CanCounter333333: CTU;
	M: INT;
	DFS: CTU;
	LINCOLN: BOOL;

	LDS: BOOL;
	DSS: BOOL;
	K: INT;
	KJSJHE: BOOL;
	PLOP: INT;
	HLJKLTFK: CTU;
	FGHJD: INT;
	CancounterM2: CTU;
	CancounterM12: CTU;
	sc_Depal1_1stshiftcount: INT;
	try: INT;
	COUNTPULSE: BOOL;
	_TEST: CTU;
	_1stshiftcc: INT;
	_2NDshiftcc: INT;
	sc_M1CCReset: BOOL;
	Pallet_Count: INT;
	EmptyCans_Initial: REAL;
	InitialPalletCount: INT:=3276;
	TESTPALLETCOUNT: CTU;
	TESTPC: INT;
	M2CanCNTPE: BOOL;
	M2CanCountPE: BOOL;
	CanCounterCTU: CTU;
	CanCountWORD: WORD;
	CanCountMultiplier: CTU;
	MultiplierWORD: WORD;
	HighCount: REAL;
	MultiplierREAL: REAL;
	CanCountREAL: REAL;
	ActualCount: REAL;
	ChainHoistDown: Toggle;
	CHainHoistUp: TOGGLE;
	Infeed1: TOGGLE;
	ElevatorInfeed: TOGGLE;
	Elevatorrev: TOGGLE;
	Infeed2: Toggle;
	Infeed2REV: Toggle;
	Infeed1REV: TOGGLE;
	ELETOggle: TOGGLE;
	Cap: TOGGLE;
	Capture: TOGGLE;
	Release: TOGGLE;
	Rel: TOGGLE;
	hsclose: TOGGLE;
	sHoistSClose: BOOL;
	ABCD: TOGGLE;
	efgh: TOGGLE;
	CarFwd: Toggle;
	CarRev: Toggle;
	sDischarge1Run: BOOL;
	Discharge1Toggle: Toggle;
	Discharge2Run: Toggle;
	sDischarge2Run: BOOL;
	GD1: BOOL;
	Verify: TON;
	SetForNewPallet: SR;
	SendCarriageBack: BOOL;
	SetCarrRev: BOOL;
	Hoist_Tog_Resets: BOOL;
END_VAR
VAR_INPUT
	ProductHeight_Pos: BOOL;
	Carriage_to_Pickup: BOOL;
	Fwd_Enable: BOOL;
	DR1_Tog: TOGGLE;


END_VAR
VAR // added by the converter: edge detectors and wires of the graphical bodies
    _w1, _w2, _w3, _w4, _w5, _w6, _w7, _w8 : BOOL;
END_VAR

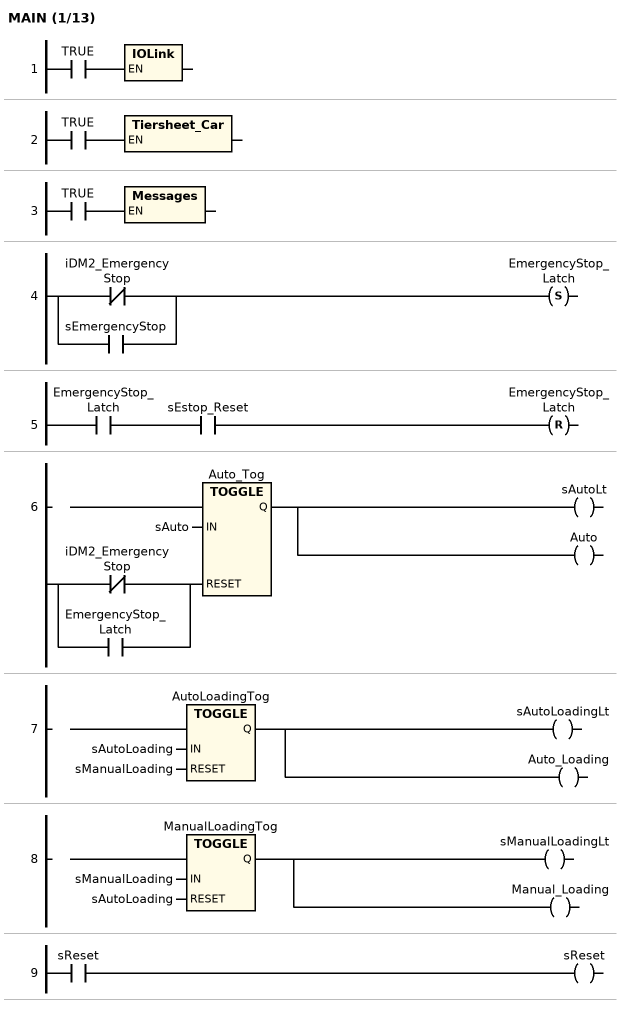
// NETWORK 1
IOLink();

// NETWORK 2
Tiersheet_Car();

// NETWORK 3
Messages();

// NETWORK 4
EmergencyStop_Latch S= NOT iDM2_EmergencyStop OR sEmergencyStop;

// NETWORK 5
EmergencyStop_Latch R= EmergencyStop_Latch AND sEstop_Reset;

// NETWORK 6
Auto_Tog(IN := sAuto, RESET := NOT iDM2_EmergencyStop OR EmergencyStop_Latch); // TOGGLE
sAutoLt := Auto_Tog.Q;
Auto := Auto_Tog.Q;

// NETWORK 7
AutoLoadingTog(IN := sAutoLoading, RESET := sManualLoading); // TOGGLE
sAutoLoadingLt := AutoLoadingTog.Q;
Auto_Loading := AutoLoadingTog.Q;

// NETWORK 8
ManualLoadingTog(IN := sManualLoading, RESET := sAutoLoading); // TOGGLE
sManualLoadingLt := ManualLoadingTog.Q;
Manual_Loading := ManualLoadingTog.Q;

// NETWORK 9
sReset := sReset;

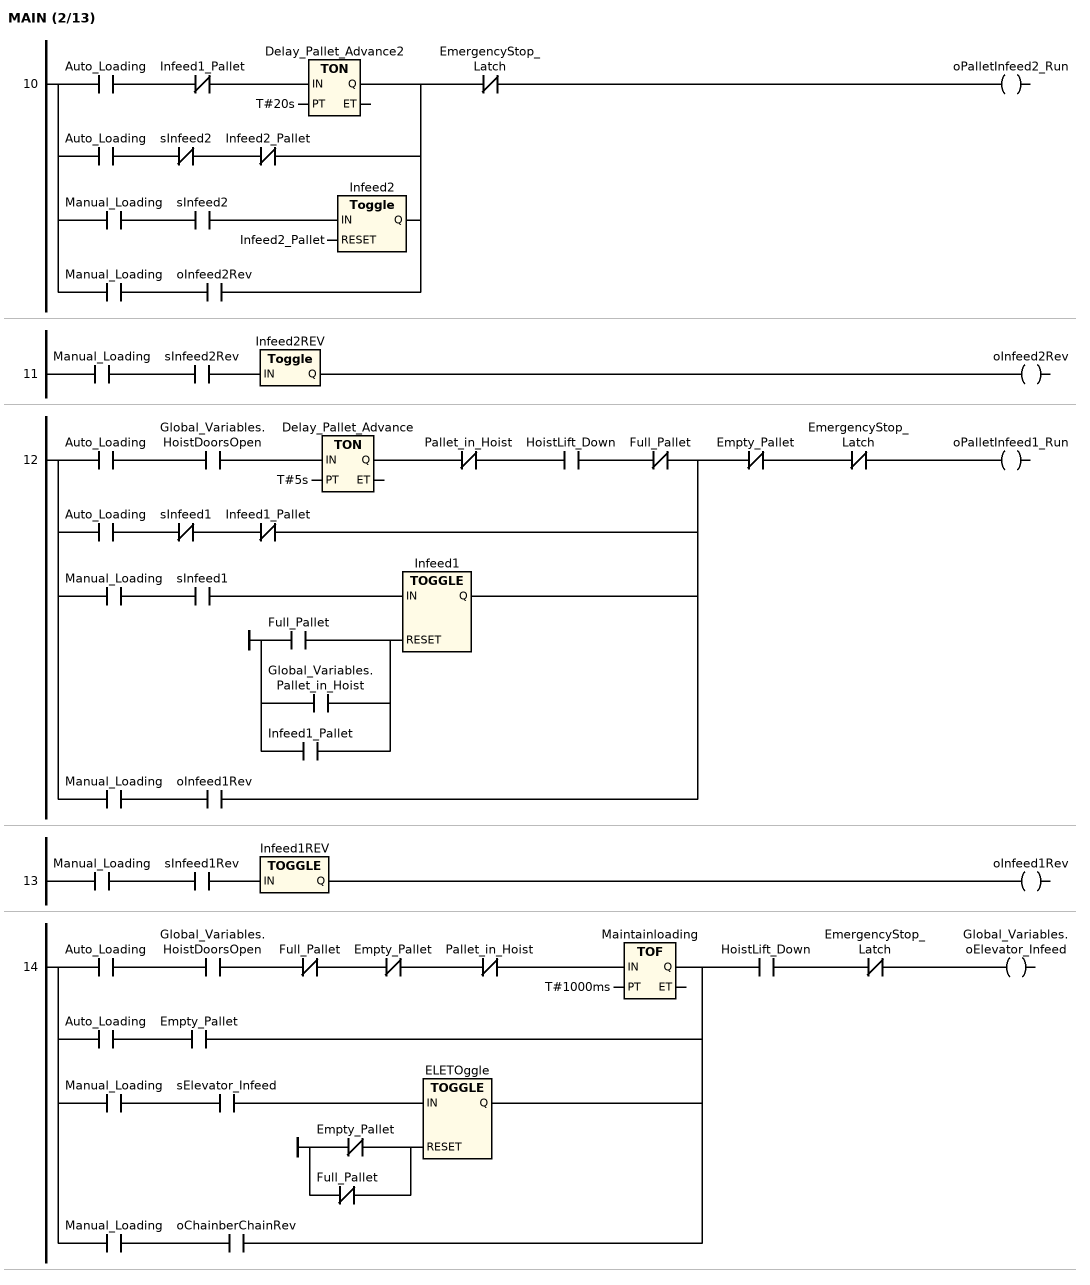
// NETWORK 10
Delay_Pallet_Advance2(IN := Auto_Loading AND NOT Infeed1_Pallet, PT := T#20s); // TON
Infeed2(IN := Manual_Loading AND sInfeed2, RESET := Infeed2_Pallet); // Toggle
oPalletInfeed2_Run := (Delay_Pallet_Advance2.Q OR Auto_Loading AND NOT sInfeed2 AND NOT Infeed2_Pallet OR Infeed2.Q OR Manual_Loading AND oInfeed2Rev) AND NOT EmergencyStop_Latch;

// NETWORK 11
Infeed2REV(IN := Manual_Loading AND sInfeed2Rev); // Toggle
oInfeed2Rev := Infeed2REV.Q;

// NETWORK 12
Delay_Pallet_Advance(IN := Auto_Loading AND Global_Variables.HoistDoorsOpen, PT := T#5s); // TON
Infeed1(IN := Manual_Loading AND sInfeed1, RESET := Full_Pallet OR Global_Variables.Pallet_in_Hoist OR Infeed1_Pallet); // TOGGLE
oPalletInfeed1_Run := (Delay_Pallet_Advance.Q AND NOT Pallet_in_Hoist AND HoistLift_Down AND NOT Full_Pallet OR Auto_Loading AND NOT sInfeed1 AND NOT Infeed1_Pallet OR Infeed1.Q OR Manual_Loading AND oInfeed1Rev) AND NOT Empty_Pallet AND NOT EmergencyStop_Latch;

// NETWORK 13
Infeed1REV(IN := Manual_Loading AND sInfeed1Rev); // TOGGLE
oInfeed1Rev := Infeed1REV.Q;

// NETWORK 14
Maintainloading(IN := Auto_Loading AND Global_Variables.HoistDoorsOpen AND NOT Full_Pallet AND NOT Empty_Pallet AND NOT Pallet_in_Hoist, PT := T#1000ms); // TOF
ELETOggle(IN := Manual_Loading AND sElevator_Infeed, RESET := NOT Empty_Pallet OR NOT Full_Pallet); // TOGGLE
Global_Variables.oElevator_Infeed := (Maintainloading.Q OR Auto_Loading AND Empty_Pallet OR ELETOggle.Q OR Manual_Loading AND oChainberChainRev) AND HoistLift_Down AND NOT EmergencyStop_Latch;

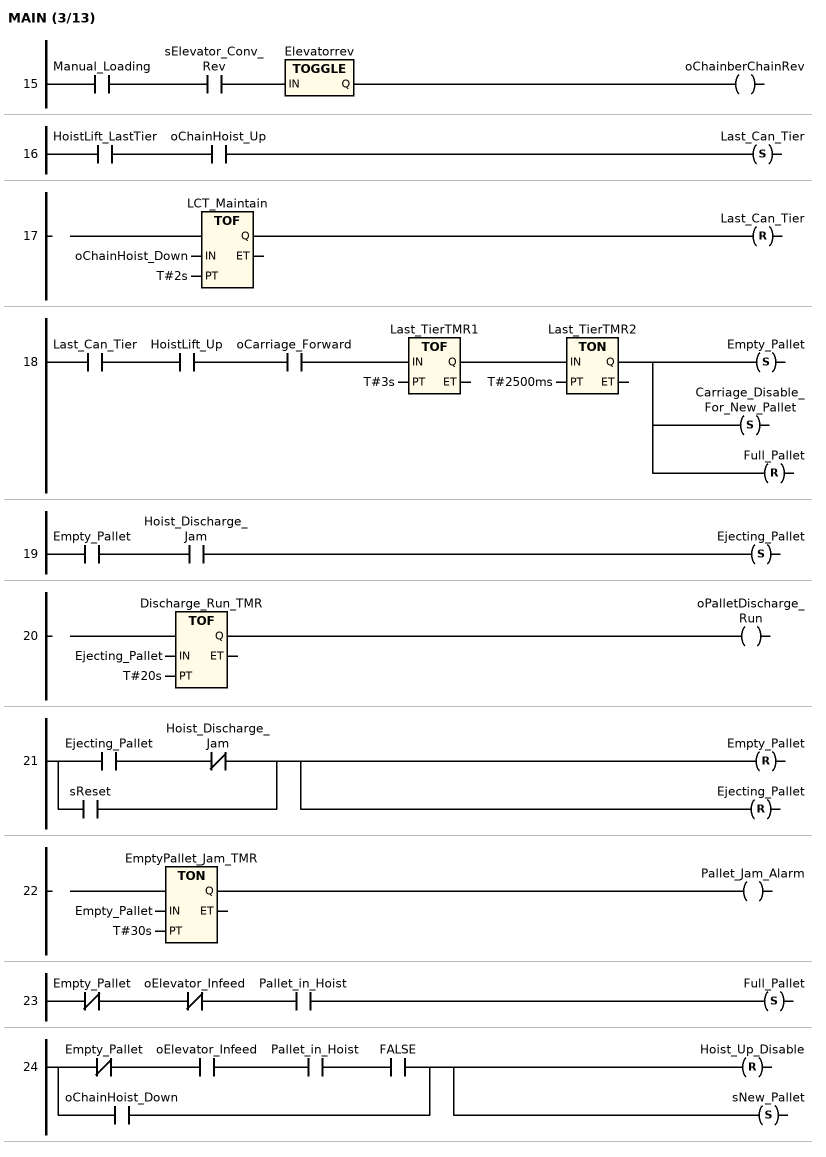
// NETWORK 15
Elevatorrev(IN := Manual_Loading AND sElevator_Conv_Rev); // TOGGLE
oChainberChainRev := Elevatorrev.Q;

// NETWORK 16
Last_Can_Tier S= HoistLift_LastTier AND oChainHoist_Up;

// NETWORK 17
LCT_Maintain(IN := oChainHoist_Down, PT := T#2s); // TOF
Last_Can_Tier R= LCT_Maintain.Q;

// NETWORK 18
Last_TierTMR1(IN := Last_Can_Tier AND HoistLift_Up AND oCarriage_Forward, PT := T#3s); // TOF
Last_TierTMR2(IN := Last_TierTMR1.Q, PT := T#2500ms); // TON
Empty_Pallet S= Last_TierTMR2.Q;
Carriage_Disable_For_New_Pallet S= Last_TierTMR2.Q;
Full_Pallet R= Last_TierTMR2.Q;

// NETWORK 19
Ejecting_Pallet S= Empty_Pallet AND Hoist_Discharge_Jam;

// NETWORK 20
Discharge_Run_TMR(IN := Ejecting_Pallet, PT := T#20s); // TOF
oPalletDischarge_Run := Discharge_Run_TMR.Q;

// NETWORK 21
_w1 := Ejecting_Pallet AND NOT Hoist_Discharge_Jam OR sReset;
Empty_Pallet R= _w1;
Ejecting_Pallet R= _w1;

// NETWORK 22
EmptyPallet_Jam_TMR(IN := Empty_Pallet, PT := T#30s); // TON
Pallet_Jam_Alarm := EmptyPallet_Jam_TMR.Q;

// NETWORK 23
Full_Pallet S= NOT Empty_Pallet AND NOT oElevator_Infeed AND Pallet_in_Hoist;

// NETWORK 24
_w2 := NOT Empty_Pallet AND oElevator_Infeed AND Pallet_in_Hoist AND FALSE OR oChainHoist_Down;
Hoist_Up_Disable R= _w2;
sNew_Pallet S= _w2;

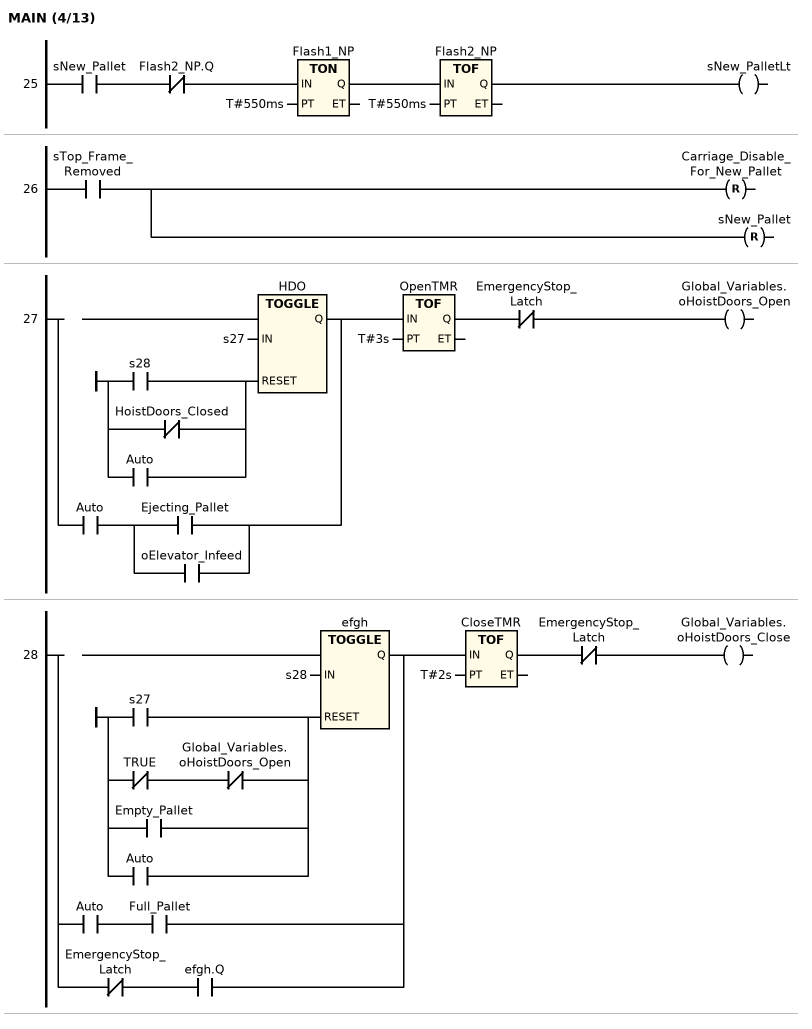
// NETWORK 25
Flash1_NP(IN := sNew_Pallet AND NOT Flash2_NP.Q, PT := T#550ms); // TON
Flash2_NP(IN := Flash1_NP.Q, PT := T#550ms); // TOF
sNew_PalletLt := Flash2_NP.Q;

// NETWORK 26
Carriage_Disable_For_New_Pallet R= sTop_Frame_Removed;
sNew_Pallet R= sTop_Frame_Removed;

// NETWORK 27
HDO(IN := s27, RESET := s28 OR NOT HoistDoors_Closed OR Auto); // TOGGLE
OpenTMR(IN := HDO.Q OR Auto AND (Ejecting_Pallet OR oElevator_Infeed), PT := T#3s); // TOF
Global_Variables.oHoistDoors_Open := OpenTMR.Q AND NOT EmergencyStop_Latch;

// NETWORK 28
efgh(IN := s28, RESET := s27 OR NOT TRUE AND NOT Global_Variables.oHoistDoors_Open OR Empty_Pallet OR Auto); // TOGGLE
CloseTMR(IN := efgh.Q OR Auto AND Full_Pallet OR NOT EmergencyStop_Latch AND efgh.Q, PT := T#2s); // TOF
Global_Variables.oHoistDoors_Close := CloseTMR.Q AND NOT EmergencyStop_Latch;

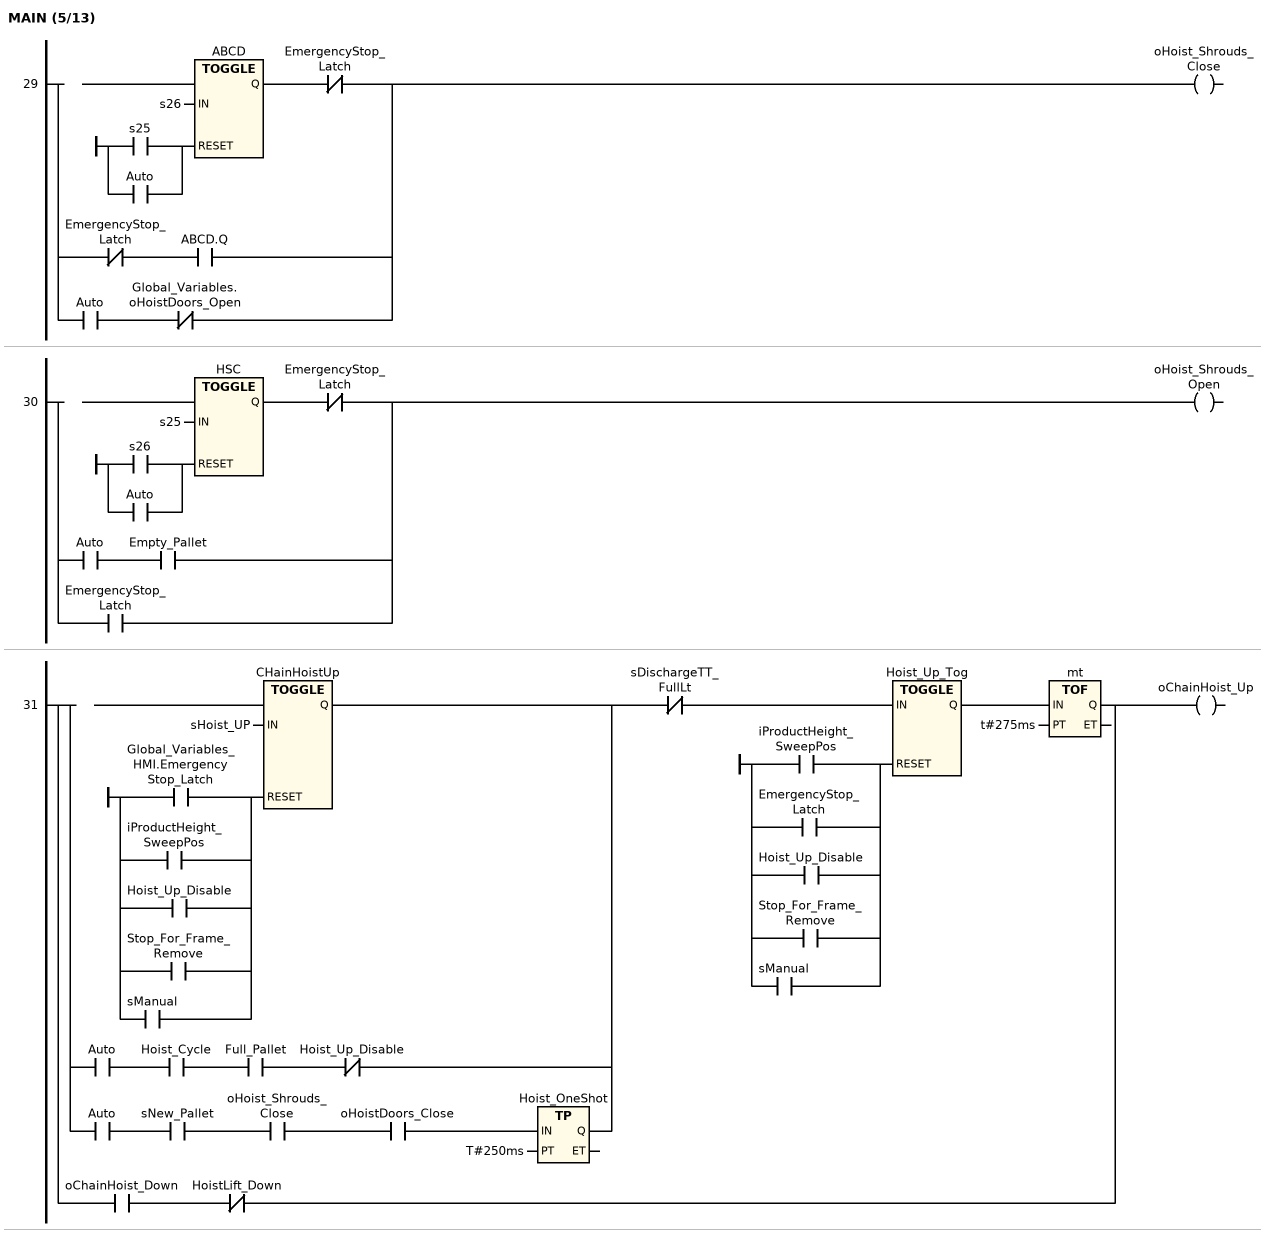
// NETWORK 29
ABCD(IN := s26, RESET := s25 OR Auto); // TOGGLE
oHoist_Shrouds_Close := ABCD.Q AND NOT EmergencyStop_Latch OR NOT EmergencyStop_Latch AND ABCD.Q OR Auto AND NOT Global_Variables.oHoistDoors_Open;

// NETWORK 30
HSC(IN := s25, RESET := s26 OR Auto); // TOGGLE
oHoist_Shrouds_Open := HSC.Q AND NOT EmergencyStop_Latch OR Auto AND Empty_Pallet OR EmergencyStop_Latch;

// NETWORK 31
CHainHoistUp(IN := sHoist_UP, RESET := Global_Variables_HMI.EmergencyStop_Latch OR iProductHeight_SweepPos OR Hoist_Up_Disable OR Stop_For_Frame_Remove OR sManual); // TOGGLE
Hoist_OneShot(IN := Auto AND sNew_Pallet AND oHoist_Shrouds_Close AND oHoistDoors_Close, PT := T#250ms); // TP
Hoist_Up_Tog(IN := (CHainHoistUp.Q OR Auto AND Hoist_Cycle AND Full_Pallet AND NOT Hoist_Up_Disable OR Hoist_OneShot.Q) AND NOT sDischargeTT_FullLt, RESET := iProductHeight_SweepPos OR EmergencyStop_Latch OR Hoist_Up_Disable OR Stop_For_Frame_Remove OR sManual); // TOGGLE
mt(IN := Hoist_Up_Tog.Q, PT := t#275ms); // TOF
oChainHoist_Up := mt.Q OR oChainHoist_Down AND NOT HoistLift_Down;

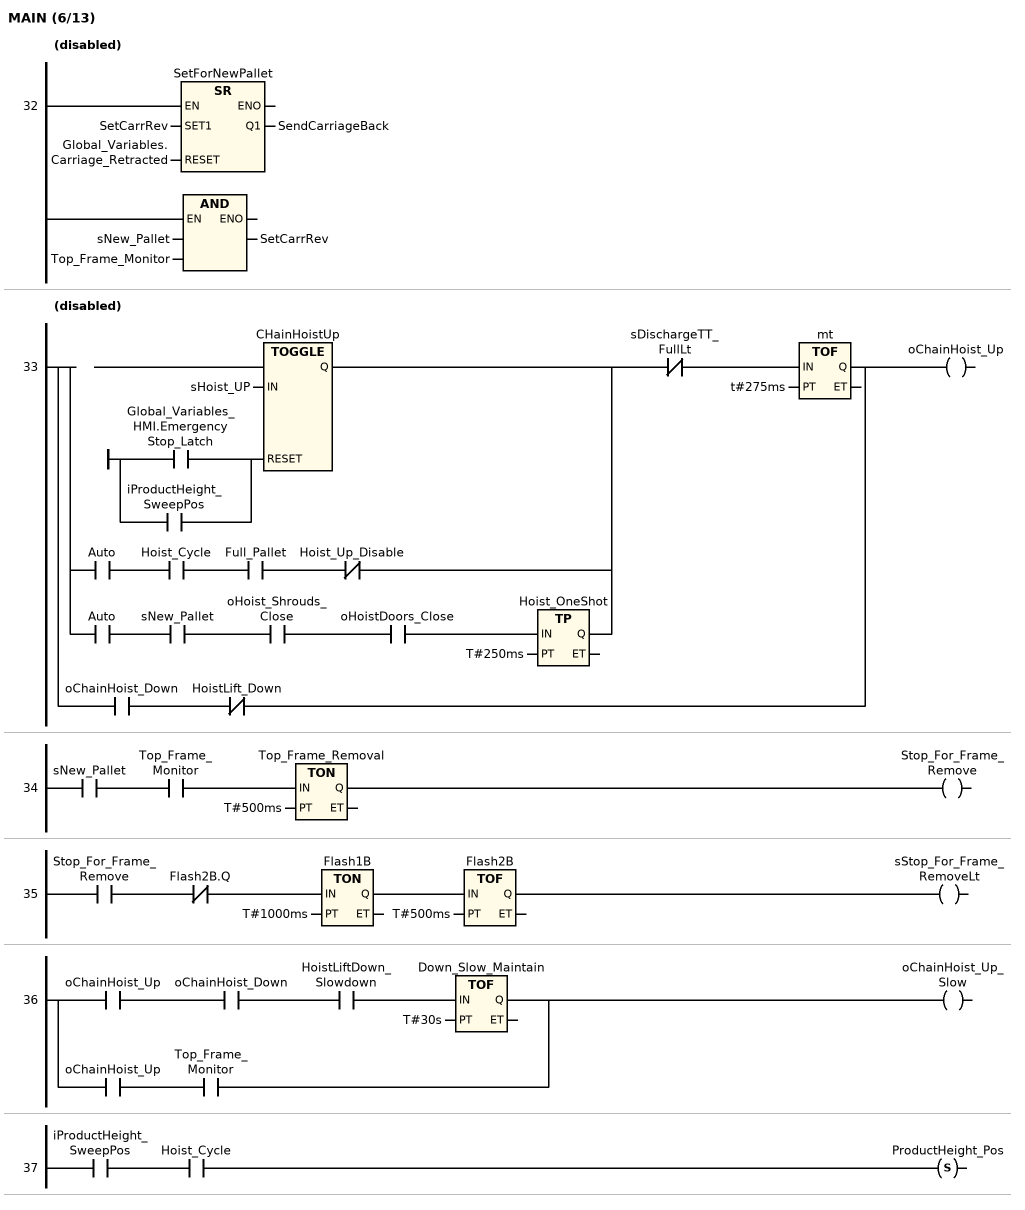
// NETWORK 32 (disabled)
// SetForNewPallet(SET1 := SetCarrRev, RESET := Global_Variables.Carriage_Retracted, Q1 => SendCarriageBack); // SR
// SetCarrRev := sNew_Pallet AND Top_Frame_Monitor;

// NETWORK 33 (disabled)
// CHainHoistUp(IN := sHoist_UP, RESET := Global_Variables_HMI.EmergencyStop_Latch OR iProductHeight_SweepPos); // TOGGLE
// Hoist_OneShot(IN := Auto AND sNew_Pallet AND oHoist_Shrouds_Close AND oHoistDoors_Close, PT := T#250ms); // TP
// mt(IN := (CHainHoistUp.Q OR Auto AND Hoist_Cycle AND Full_Pallet AND NOT Hoist_Up_Disable OR Hoist_OneShot.Q) AND NOT sDischargeTT_FullLt, PT := t#275ms); // TOF
// oChainHoist_Up := mt.Q OR oChainHoist_Down AND NOT HoistLift_Down;

// NETWORK 34
Top_Frame_Removal(IN := sNew_Pallet AND Top_Frame_Monitor, PT := T#500ms); // TON
Stop_For_Frame_Remove := Top_Frame_Removal.Q;

// NETWORK 35
Flash1B(IN := Stop_For_Frame_Remove AND NOT Flash2B.Q, PT := T#1000ms); // TON
Flash2B(IN := Flash1B.Q, PT := T#500ms); // TOF
sStop_For_Frame_RemoveLt := Flash2B.Q;

// NETWORK 36
Down_Slow_Maintain(IN := oChainHoist_Up AND (oChainHoist_Down AND HoistLiftDown_Slowdown), PT := T#30s); // TOF
oChainHoist_Up_Slow := Down_Slow_Maintain.Q OR oChainHoist_Up AND Top_Frame_Monitor;

// NETWORK 37
ProductHeight_Pos S= iProductHeight_SweepPos AND Hoist_Cycle;

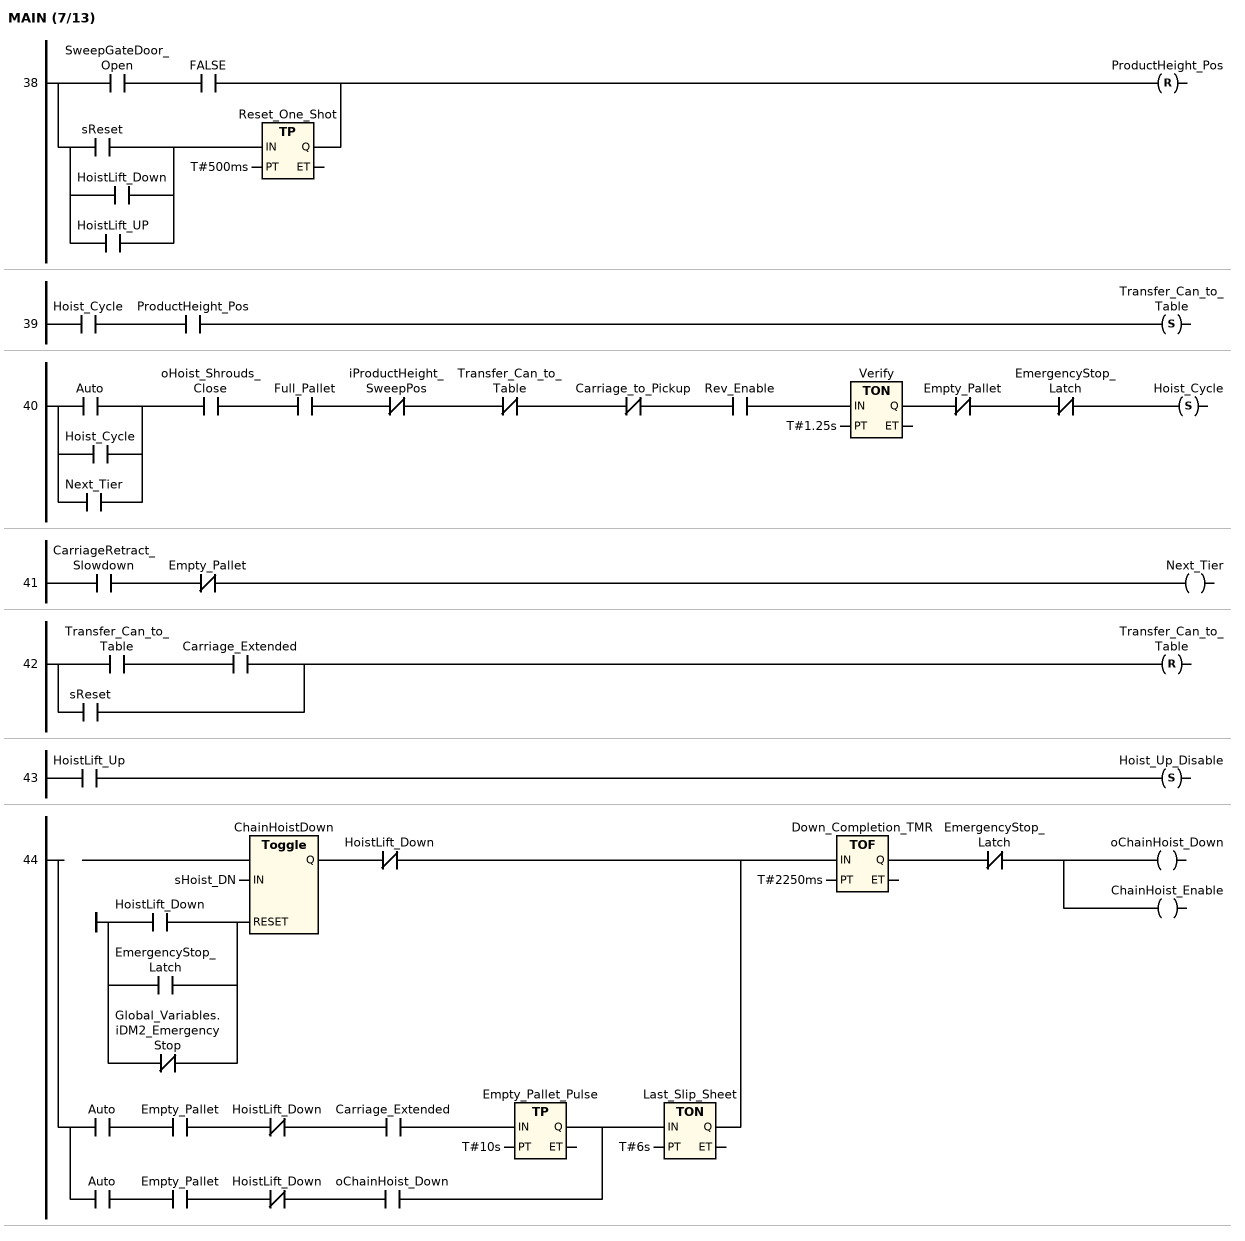
// NETWORK 38
Reset_One_Shot(IN := sReset OR HoistLift_Down OR HoistLift_UP, PT := T#500ms); // TP
ProductHeight_Pos R= SweepGateDoor_Open AND FALSE OR Reset_One_Shot.Q;

// NETWORK 39
Transfer_Can_to_Table S= Hoist_Cycle AND ProductHeight_Pos;

// NETWORK 40
Verify(IN := (Auto OR Hoist_Cycle OR Next_Tier) AND oHoist_Shrouds_Close AND Full_Pallet AND NOT iProductHeight_SweepPos AND NOT Transfer_Can_to_Table AND NOT Carriage_to_Pickup AND Rev_Enable, PT := T#1.25s); // TON
Hoist_Cycle S= Verify.Q AND NOT Empty_Pallet AND NOT EmergencyStop_Latch;

// NETWORK 41
Next_Tier := CarriageRetract_Slowdown AND NOT Empty_Pallet;

// NETWORK 42
Transfer_Can_to_Table R= Transfer_Can_to_Table AND Carriage_Extended OR sReset;

// NETWORK 43
Hoist_Up_Disable S= HoistLift_Up;

// NETWORK 44
ChainHoistDown(IN := sHoist_DN, RESET := HoistLift_Down OR EmergencyStop_Latch OR NOT Global_Variables.iDM2_EmergencyStop); // Toggle
Empty_Pallet_Pulse(IN := Auto AND Empty_Pallet AND NOT HoistLift_Down AND Carriage_Extended, PT := T#10s); // TP
Last_Slip_Sheet(IN := Empty_Pallet_Pulse.Q OR Auto AND Empty_Pallet AND NOT HoistLift_Down AND oChainHoist_Down, PT := T#6s); // TON
Down_Completion_TMR(IN := ChainHoistDown.Q AND NOT HoistLift_Down OR Last_Slip_Sheet.Q, PT := T#2250ms); // TOF
_w3 := Down_Completion_TMR.Q AND NOT EmergencyStop_Latch;
oChainHoist_Down := _w3;
ChainHoist_Enable := _w3;

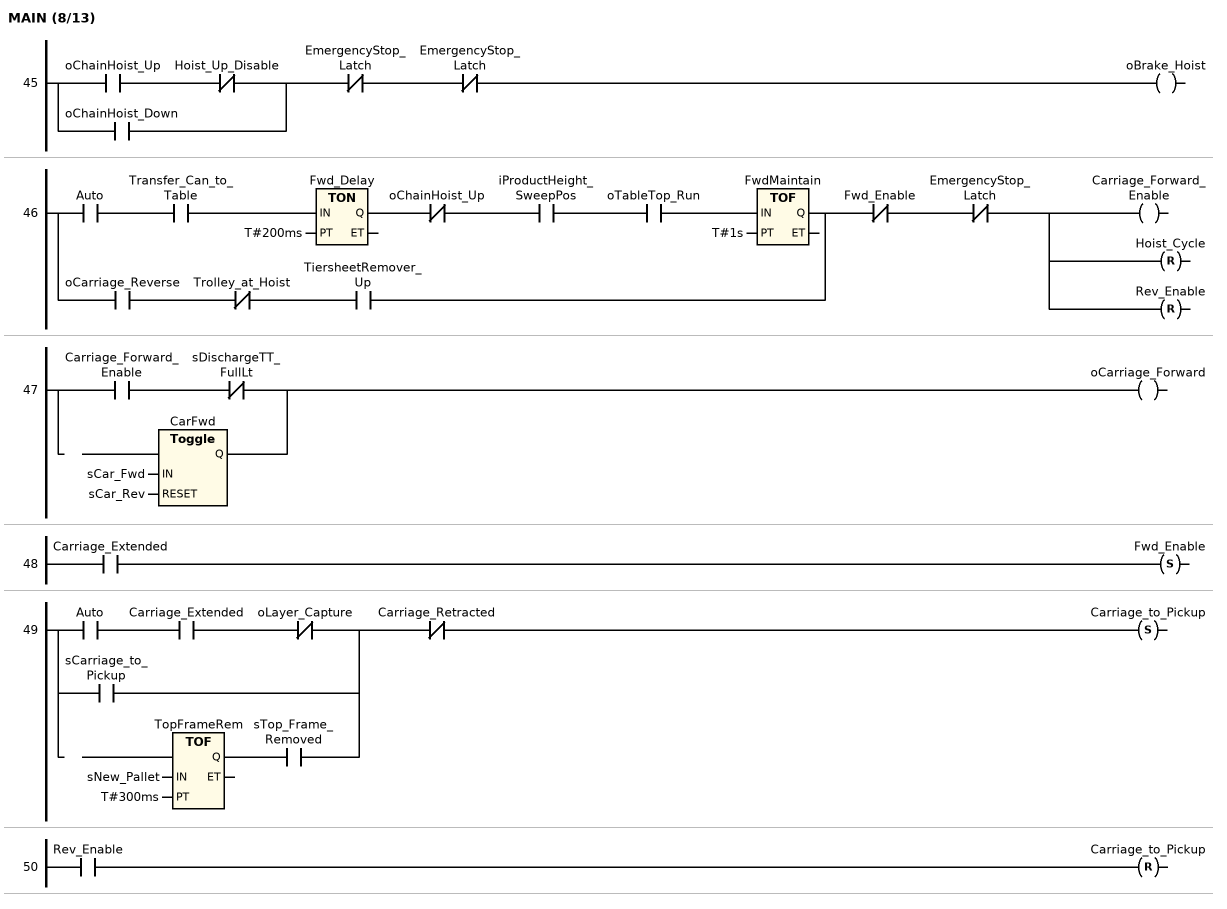
// NETWORK 45
oBrake_Hoist := (oChainHoist_Up AND NOT Hoist_Up_Disable OR oChainHoist_Down) AND NOT EmergencyStop_Latch AND NOT EmergencyStop_Latch;

// NETWORK 46
Fwd_Delay(IN := Auto AND Transfer_Can_to_Table, PT := T#200ms); // TON
FwdMaintain(IN := Fwd_Delay.Q AND NOT oChainHoist_Up AND iProductHeight_SweepPos AND oTableTop_Run, PT := T#1s); // TOF
_w4 := (FwdMaintain.Q OR oCarriage_Reverse AND NOT Trolley_at_Hoist AND TiersheetRemover_Up) AND NOT Fwd_Enable AND NOT EmergencyStop_Latch;
Carriage_Forward_Enable := _w4;
Hoist_Cycle R= _w4;
Rev_Enable R= _w4;

// NETWORK 47
CarFwd(IN := sCar_Fwd, RESET := sCar_Rev); // Toggle
oCarriage_Forward := Carriage_Forward_Enable AND NOT sDischargeTT_FullLt OR CarFwd.Q;

// NETWORK 48
Fwd_Enable S= Carriage_Extended;

// NETWORK 49
TopFrameRem(IN := sNew_Pallet, PT := T#300ms); // TOF
Carriage_to_Pickup S= (Auto AND Carriage_Extended AND NOT oLayer_Capture OR sCarriage_to_Pickup OR TopFrameRem.Q AND sTop_Frame_Removed) AND NOT Carriage_Retracted;

// NETWORK 50
Carriage_to_Pickup R= Rev_Enable;

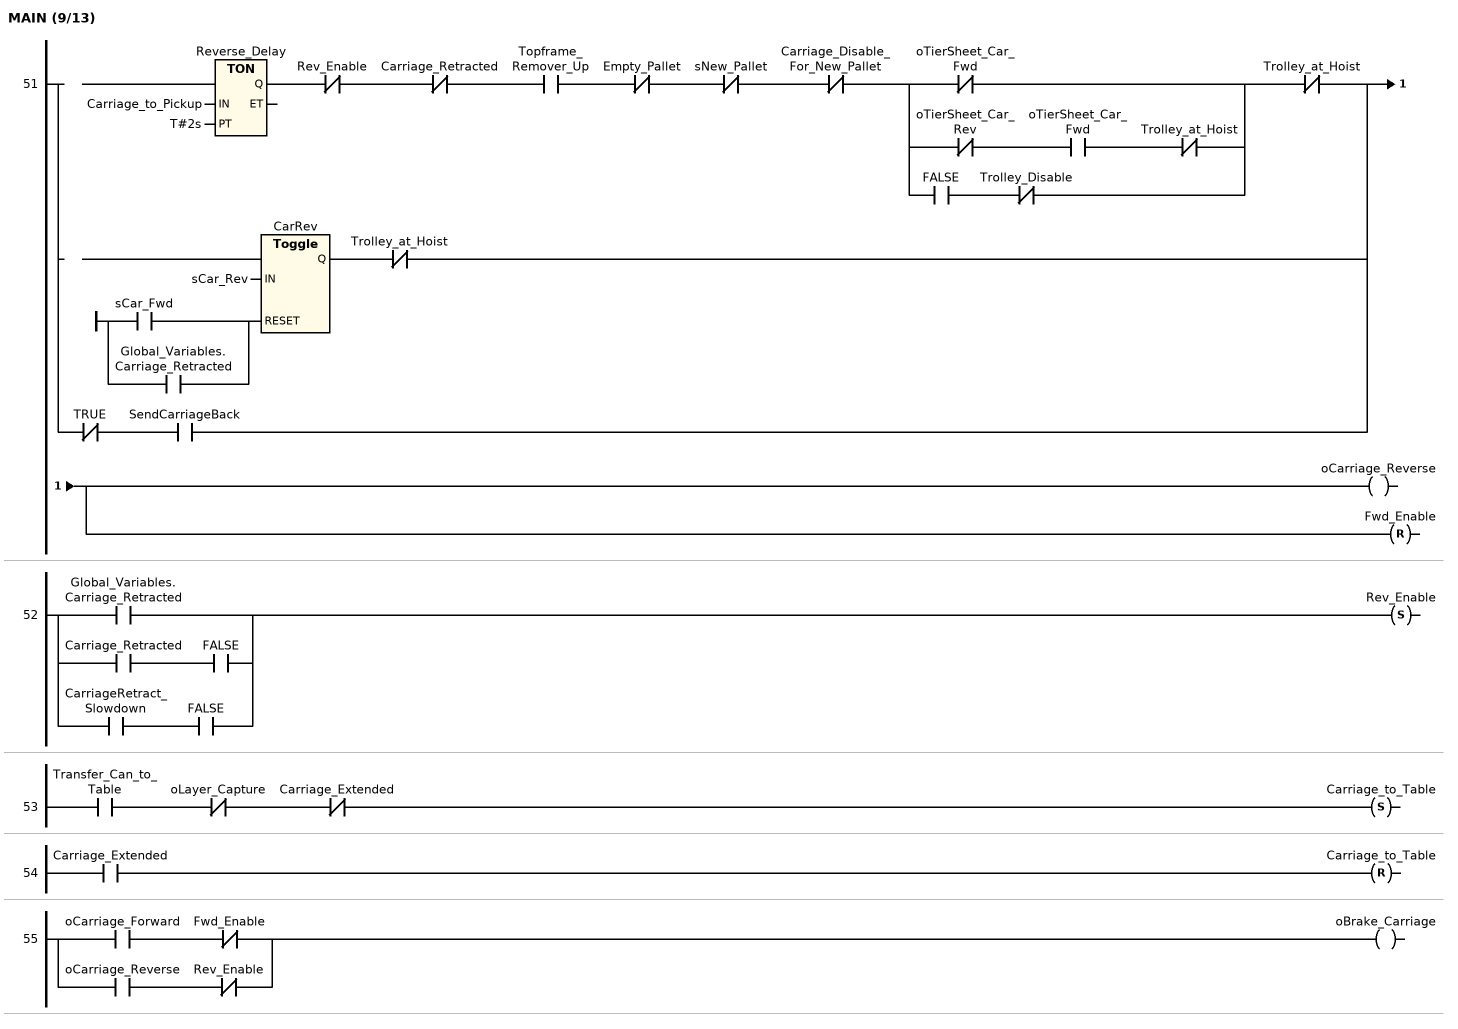
// NETWORK 51
Reverse_Delay(IN := Carriage_to_Pickup, PT := T#2s); // TON
CarRev(IN := sCar_Rev, RESET := sCar_Fwd OR Global_Variables.Carriage_Retracted); // Toggle
_w5 := Reverse_Delay.Q AND NOT Rev_Enable AND NOT Carriage_Retracted AND Topframe_Remover_Up AND NOT Empty_Pallet AND NOT sNew_Pallet AND NOT Carriage_Disable_For_New_Pallet AND (NOT oTierSheet_Car_Fwd OR NOT oTierSheet_Car_Rev AND oTierSheet_Car_Fwd AND NOT Trolley_at_Hoist OR FALSE AND NOT Trolley_Disable) AND NOT Trolley_at_Hoist OR CarRev.Q AND NOT Trolley_at_Hoist OR NOT TRUE AND SendCarriageBack;
oCarriage_Reverse := _w5;
Fwd_Enable R= _w5;

// NETWORK 52
Rev_Enable S= Global_Variables.Carriage_Retracted OR Carriage_Retracted AND FALSE OR CarriageRetract_Slowdown AND FALSE;

// NETWORK 53
Carriage_to_Table S= Transfer_Can_to_Table AND NOT oLayer_Capture AND NOT Carriage_Extended;

// NETWORK 54
Carriage_to_Table R= Carriage_Extended;

// NETWORK 55
oBrake_Carriage := oCarriage_Forward AND NOT Fwd_Enable OR oCarriage_Reverse AND NOT Rev_Enable;

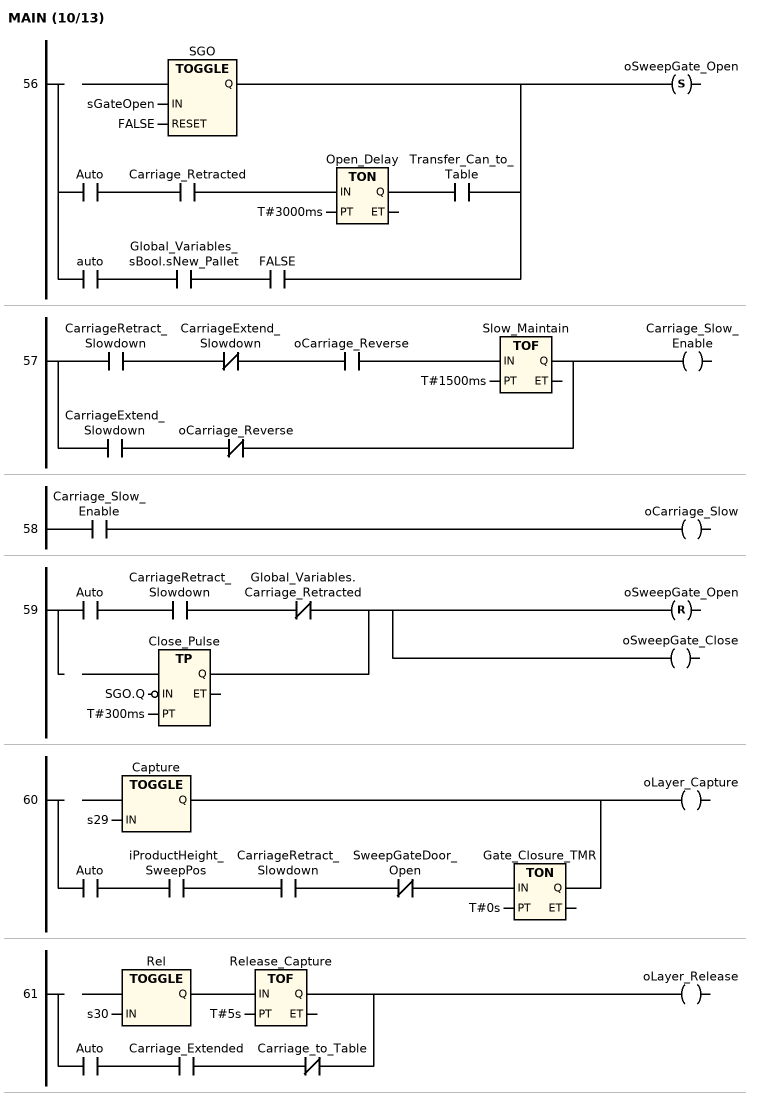
// NETWORK 56
SGO(IN := sGateOpen, RESET := FALSE); // TOGGLE
Open_Delay(IN := Auto AND Carriage_Retracted, PT := T#3000ms); // TON
oSweepGate_Open S= SGO.Q OR Open_Delay.Q AND Transfer_Can_to_Table OR auto AND Global_Variables_sBool.sNew_Pallet AND FALSE;

// NETWORK 57
Slow_Maintain(IN := CarriageRetract_Slowdown AND NOT CarriageExtend_Slowdown AND oCarriage_Reverse, PT := T#1500ms); // TOF
Carriage_Slow_Enable := Slow_Maintain.Q OR CarriageExtend_Slowdown AND NOT oCarriage_Reverse;

// NETWORK 58
oCarriage_Slow := Carriage_Slow_Enable;

// NETWORK 59
Close_Pulse(IN := NOT SGO.Q, PT := T#300ms); // TP
_w6 := Auto AND CarriageRetract_Slowdown AND NOT Global_Variables.Carriage_Retracted OR Close_Pulse.Q;
oSweepGate_Open R= _w6;
oSweepGate_Close := _w6;

// NETWORK 60
Capture(IN := s29); // TOGGLE
Gate_Closure_TMR(IN := Auto AND iProductHeight_SweepPos AND CarriageRetract_Slowdown AND NOT SweepGateDoor_Open, PT := T#0s); // TON
oLayer_Capture := Capture.Q OR Gate_Closure_TMR.Q;

// NETWORK 61
Rel(IN := s30); // TOGGLE
Release_Capture(IN := Rel.Q, PT := T#5s); // TOF
oLayer_Release := Release_Capture.Q OR Auto AND Carriage_Extended AND NOT Carriage_to_Table;

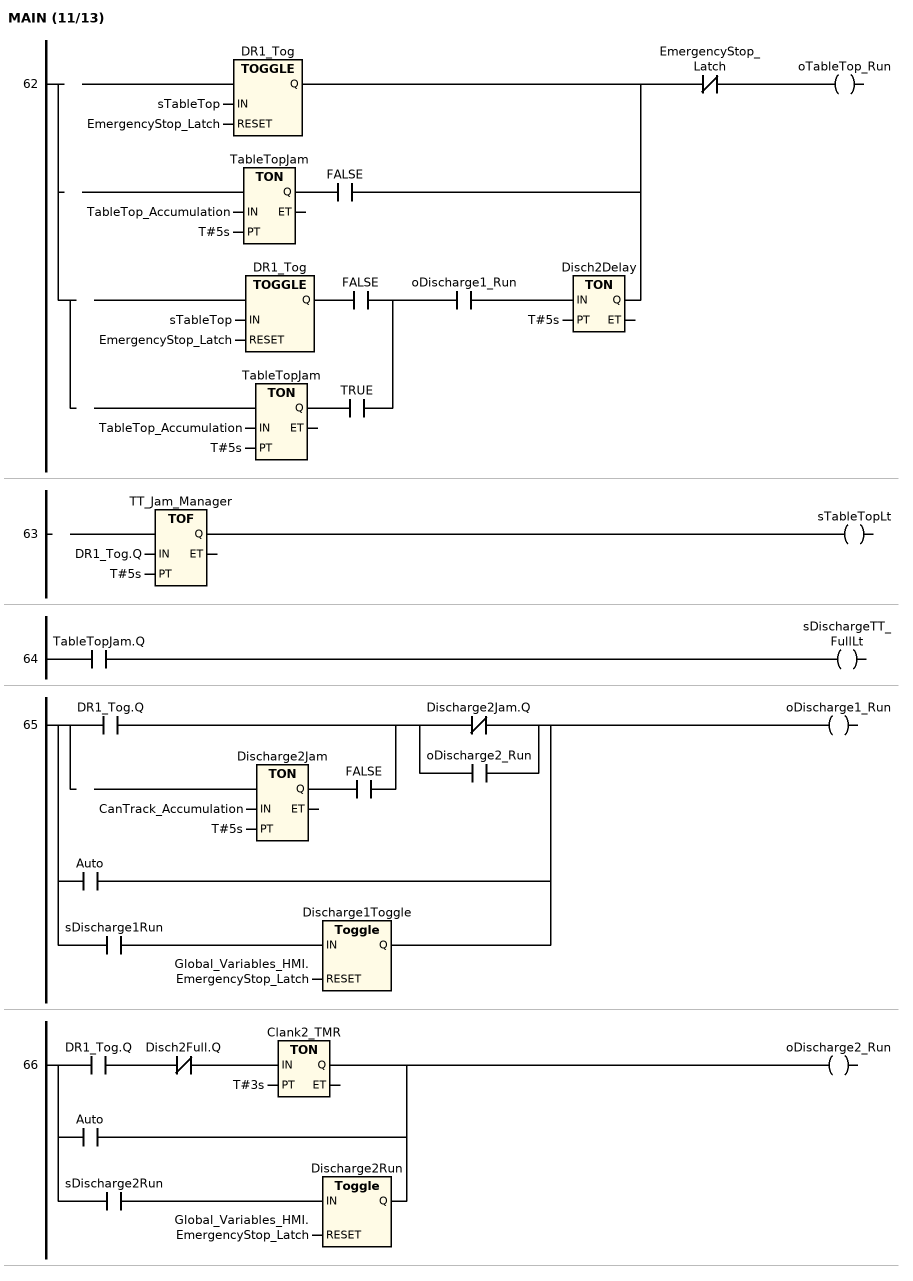
// NETWORK 62
DR1_Tog(IN := sTableTop, RESET := EmergencyStop_Latch); // TOGGLE
_w8 := DR1_Tog.Q;
TableTopJam(IN := TableTop_Accumulation, PT := T#5s); // TON
_w7 := TableTopJam.Q AND FALSE;
DR1_Tog(IN := sTableTop, RESET := EmergencyStop_Latch); // TOGGLE
TableTopJam(IN := TableTop_Accumulation, PT := T#5s); // TON
Disch2Delay(IN := (DR1_Tog.Q AND FALSE OR TableTopJam.Q AND TRUE) AND oDischarge1_Run, PT := T#5s); // TON
oTableTop_Run := (_w8 OR _w7 OR Disch2Delay.Q) AND NOT EmergencyStop_Latch;

// NETWORK 63
TT_Jam_Manager(IN := DR1_Tog.Q, PT := T#5s); // TOF
sTableTopLt := TT_Jam_Manager.Q;

// NETWORK 64
sDischargeTT_FullLt := TableTopJam.Q;

// NETWORK 65
Discharge2Jam(IN := CanTrack_Accumulation, PT := T#5s); // TON
Discharge1Toggle(IN := sDischarge1Run, RESET := Global_Variables_HMI.EmergencyStop_Latch); // Toggle
oDischarge1_Run := (DR1_Tog.Q OR Discharge2Jam.Q AND FALSE) AND (NOT Discharge2Jam.Q OR oDischarge2_Run) OR Auto OR Discharge1Toggle.Q;

// NETWORK 66
Clank2_TMR(IN := DR1_Tog.Q AND NOT Disch2Full.Q, PT := T#3s); // TON
Discharge2Run(IN := sDischarge2Run, RESET := Global_Variables_HMI.EmergencyStop_Latch); // Toggle
oDischarge2_Run := Clank2_TMR.Q OR Auto OR Discharge2Run.Q;

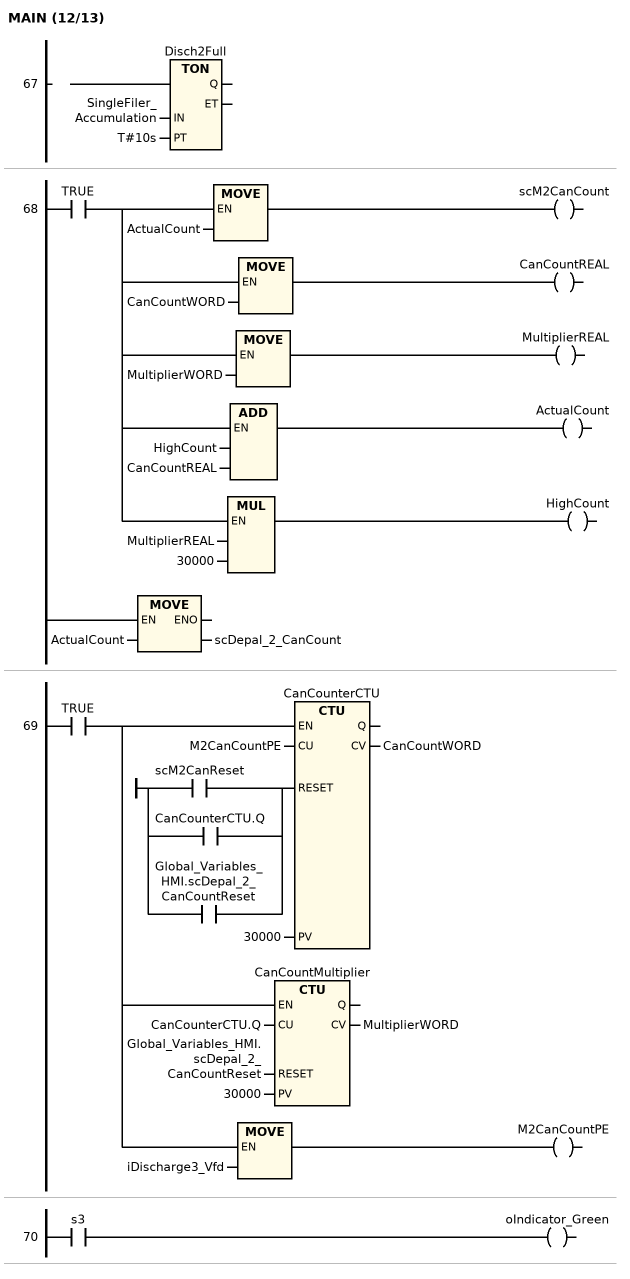
// NETWORK 67
Disch2Full(IN := SingleFiler_Accumulation, PT := T#10s); // TON

// NETWORK 68
scM2CanCount := ActualCount;
CanCountREAL := CanCountWORD;
MultiplierREAL := MultiplierWORD;
ActualCount := HighCount + CanCountREAL;
HighCount := MultiplierREAL * 30000;
scDepal_2_CanCount := ActualCount;

// NETWORK 69
CanCounterCTU(
    CU := M2CanCountPE,
    RESET := scM2CanReset OR CanCounterCTU.Q OR Global_Variables_HMI.scDepal_2_CanCountReset,
    PV := 30000,
    CV => CanCountWORD); // CTU
CanCountMultiplier(
    CU := CanCounterCTU.Q,
    RESET := Global_Variables_HMI.scDepal_2_CanCountReset,
    PV := 30000,
    CV => MultiplierWORD); // CTU
M2CanCountPE := iDischarge3_Vfd;

// NETWORK 70
oIndicator_Green := s3;

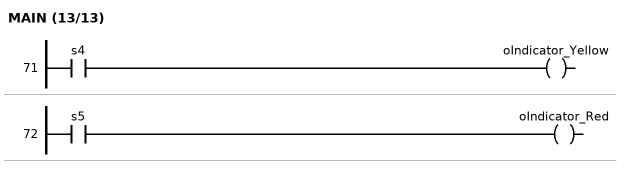
// NETWORK 71
oIndicator_Yellow := s4;

// NETWORK 72
oIndicator_Red := s5;

END_PROGRAM

// ---- POUs/Function Blocks/TOGGLE.TcPOU
FUNCTION_BLOCK TOGGLE
VAR_INPUT
	IN : BOOL;
	RESET : BOOL;
END_VAR
VAR_OUTPUT
	Q : BOOL;
END_VAR
VAR
	edge : BOOL;
END_VAR

(* This function block toggle the state of the output (Q) when the input (IN)
	transitions from a FALSE to TRUE.
	If the reset input (RESET) is true, then the output is always false *)
IF RESET THEN
	Q:=0;
ELSIF IN AND NOT edge THEN
	Q:=NOT Q;
END_IF;
edge:=IN;

END_FUNCTION_BLOCK

// ---- POUs/IOLink.TcPOU
PROGRAM IOLink
VAR


	Spare: BOOL;

	TiersheetRemoverUP: SR;
	SheetRemoverUP: BOOL;
	TiersheetCarriage_Auto: BOOL;
	Remove_Dn_TMR: TON;
END_VAR

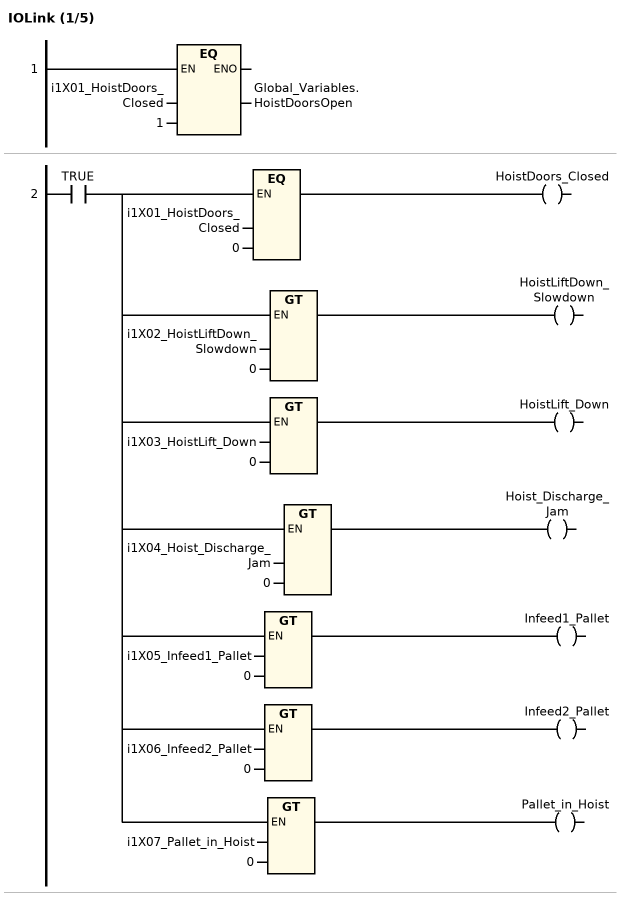
// NETWORK 1
Global_Variables.HoistDoorsOpen := i1X01_HoistDoors_Closed = 1;

// NETWORK 2
HoistDoors_Closed := i1X01_HoistDoors_Closed = 0;
HoistLiftDown_Slowdown := i1X02_HoistLiftDown_Slowdown > 0;
HoistLift_Down := i1X03_HoistLift_Down > 0;
Hoist_Discharge_Jam := i1X04_Hoist_Discharge_Jam > 0;
Infeed1_Pallet := i1X05_Infeed1_Pallet > 0;
Infeed2_Pallet := i1X06_Infeed2_Pallet > 0;
Pallet_in_Hoist := i1X07_Pallet_in_Hoist > 0;

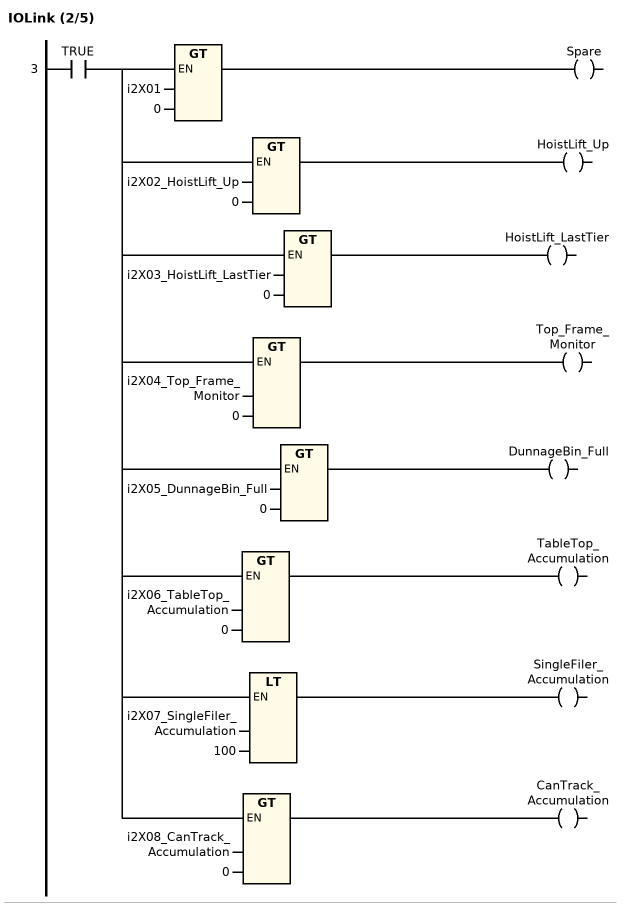
// NETWORK 3
Spare := i2X01 > 0;
HoistLift_Up := i2X02_HoistLift_Up > 0;
HoistLift_LastTier := i2X03_HoistLift_LastTier > 0;
Top_Frame_Monitor := i2X04_Top_Frame_Monitor > 0;
DunnageBin_Full := i2X05_DunnageBin_Full > 0;
TableTop_Accumulation := i2X06_TableTop_Accumulation > 0;
SingleFiler_Accumulation := i2X07_SingleFiler_Accumulation < 100;
CanTrack_Accumulation := i2X08_CanTrack_Accumulation > 0;

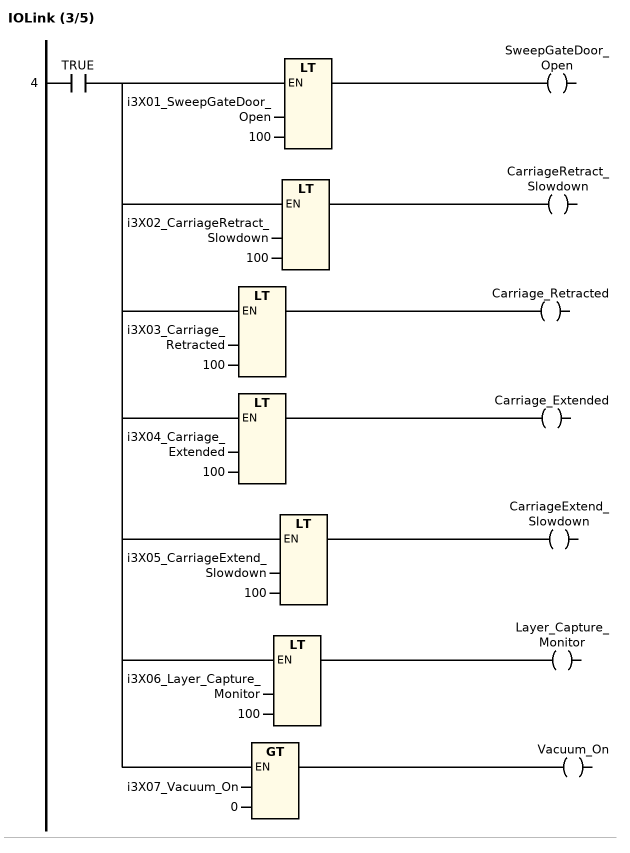
// NETWORK 4
SweepGateDoor_Open := i3X01_SweepGateDoor_Open < 100;
CarriageRetract_Slowdown := i3X02_CarriageRetract_Slowdown < 100;
Carriage_Retracted := i3X03_Carriage_Retracted < 100;
Carriage_Extended := i3X04_Carriage_Extended < 100;
CarriageExtend_Slowdown := i3X05_CarriageExtend_Slowdown < 100;
Layer_Capture_Monitor := i3X06_Layer_Capture_Monitor < 100;
Vacuum_On := i3X07_Vacuum_On > 0;

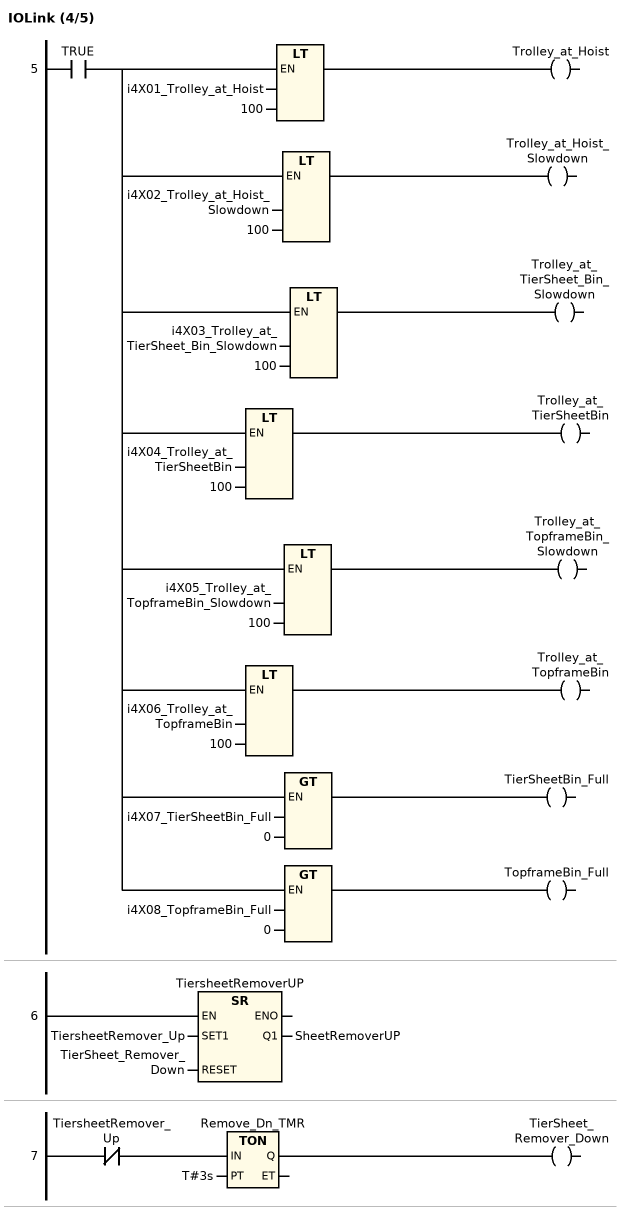
// NETWORK 5
Trolley_at_Hoist := i4X01_Trolley_at_Hoist < 100;
Trolley_at_Hoist_Slowdown := i4X02_Trolley_at_Hoist_Slowdown < 100;
Trolley_at_TierSheet_Bin_Slowdown := i4X03_Trolley_at_TierSheet_Bin_Slowdown < 100;
Trolley_at_TierSheetBin := i4X04_Trolley_at_TierSheetBin < 100;
Trolley_at_TopframeBin_Slowdown := i4X05_Trolley_at_TopframeBin_Slowdown < 100;
Trolley_at_TopframeBin := i4X06_Trolley_at_TopframeBin < 100;
TierSheetBin_Full := i4X07_TierSheetBin_Full > 0;
TopframeBin_Full := i4X08_TopframeBin_Full > 0;

// NETWORK 6
TiersheetRemoverUP(SET1 := TiersheetRemover_Up, RESET := TierSheet_Remover_Down, Q1 => SheetRemoverUP); // SR

// NETWORK 7
Remove_Dn_TMR(IN := NOT TiersheetRemover_Up, PT := T#3s); // TON
TierSheet_Remover_Down := Remove_Dn_TMR.Q;

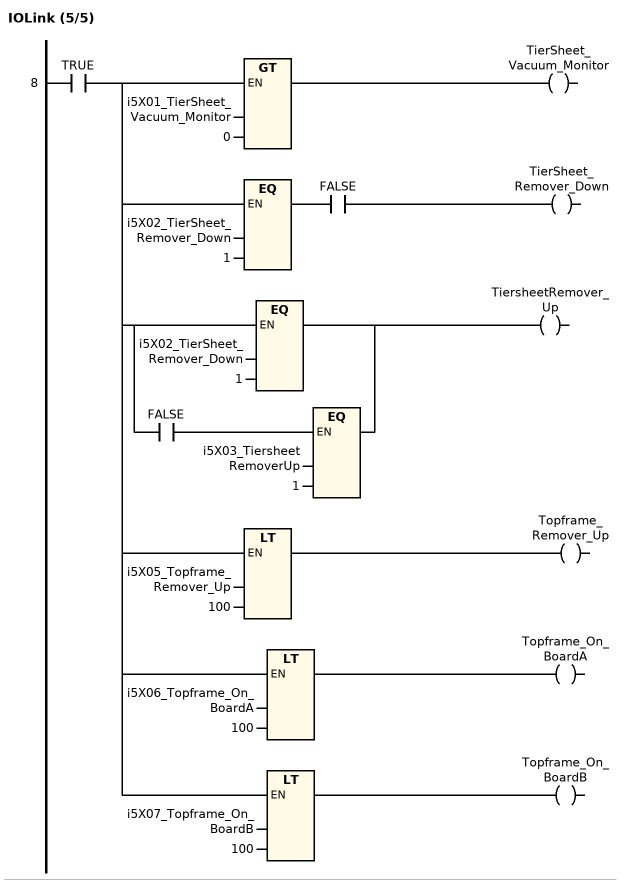
// NETWORK 8
TierSheet_Vacuum_Monitor := i5X01_TierSheet_Vacuum_Monitor > 0;
TierSheet_Remover_Down := i5X02_TierSheet_Remover_Down = 1 AND FALSE;
TiersheetRemover_Up := i5X02_TierSheet_Remover_Down = 1 OR TRUE AND FALSE AND i5X03_TiersheetRemoverUp = 1;
Topframe_Remover_Up := i5X05_Topframe_Remover_Up < 100;
Topframe_On_BoardA := i5X06_Topframe_On_BoardA < 100;
Topframe_On_BoardB := i5X07_Topframe_On_BoardB < 100;

END_PROGRAM

// ---- POUs/Tiersheet_Car.TcPOU
PROGRAM Tiersheet_Car
VAR
	TiersheetRemoverTMR: TOF;
	TrolleySlowUnlatch: TOF;
	VacTog: TOGGLE;
	SGE: TOGGLE;
	SGR: TOGGLE;

	TrolleyToSheetBin_F: BOOL;
	TrolleyToHoist_FR: BOOL;
	TrolleyToSheetBin_FR: BOOL;
	TrolleyToFrameBin_F: BOOL;
	TrolleytoHoist: BOOL;
	TrolleytoSheetBin: BOOL;
	TrolleytoFrameBin: BOOL;
	TiersheetCarriage_Auto: BOOL;
	sCarriageAuto: BOOL;
	TierCar_Tog: TOGGLE;
	sCurrent_Loc: REAL;
	sRequested_Loc: REAL;
	TrolleytoHoistSlowdown: BOOL;
	On_Loc: BOOL;
	Direction: BOOL;
	Reverse: BOOL;
	Forward: BOOL;
	t1: BOOL;
	t2: BOOL;
	t3: BOOL;
	t4: BOOL;
	t5: BOOL;
	t6: BOOL;
	L6: BOOL;
	L4: BOOL;
	L2: BOOL;
	L1: BOOL;
	Slow: BOOL;
	SlowR: BOOL;
	vactest: BOOL;
	Routine_Move_HoistToBin: BOOL;
	TiersheetRemoverTMR2: TOF;
	HoistToBin_Delay: TON;

	FrameRemover_TOG: TOGGLE;
	FrameRemoverPulse: TP;

	FrameClampsTOG: TOGGLE;
	FrameClampPulse: TP;


	At_TopFrame: BOOL;
	Gripper_Release_Pulse: TP;
	Gripper_Release_Delay: TON;
	ToSheetBinDelay: TON;

	TopFrame_Removal: BOOL;
	FrameLockPulse: TP;
	ToFrameBinDelay: TON;
	ToSheetBinDelay2: TON;




	Frame_PickUp: BOOL;
	Removal_Pulse: TP;
	Release_Delay: TON;


	Carriage_Extended_Latch: BOOL;
	Test: BOOL;
	Trolly_Delay: TON;
	TestTroley: Toggle;
	Delay: TON;
	sbTest: BOOL;
END_VAR
VAR // added by the converter: edge detectors and wires of the graphical bodies
    _w1, _w2, _w3, _w4, _w5, _w6, _w7, _w8, _w9 : INT;
    _w10, _w11 : BOOL;
END_VAR

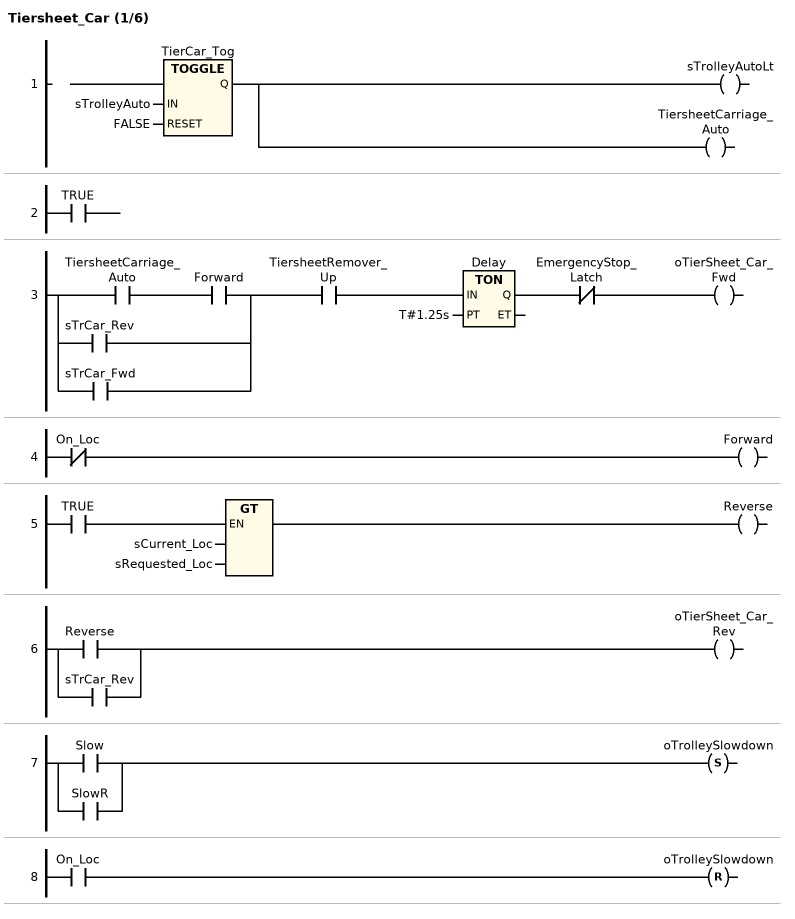
// NETWORK 1
TierCar_Tog(IN := sTrolleyAuto, RESET := FALSE); // TOGGLE
sTrolleyAutoLt := TierCar_Tog.Q;
TiersheetCarriage_Auto := TierCar_Tog.Q;

// NETWORK 2

// NETWORK 3
Delay(IN := (TiersheetCarriage_Auto AND Forward OR sTrCar_Rev OR sTrCar_Fwd) AND TiersheetRemover_Up, PT := T#1.25s); // TON
oTierSheet_Car_Fwd := Delay.Q AND NOT EmergencyStop_Latch;

// NETWORK 4
Forward := NOT On_Loc;

// NETWORK 5
Reverse := sCurrent_Loc > sRequested_Loc;

// NETWORK 6
oTierSheet_Car_Rev := Reverse OR sTrCar_Rev;

// NETWORK 7
oTrolleySlowdown S= Slow OR SlowR;

// NETWORK 8
oTrolleySlowdown R= On_Loc;

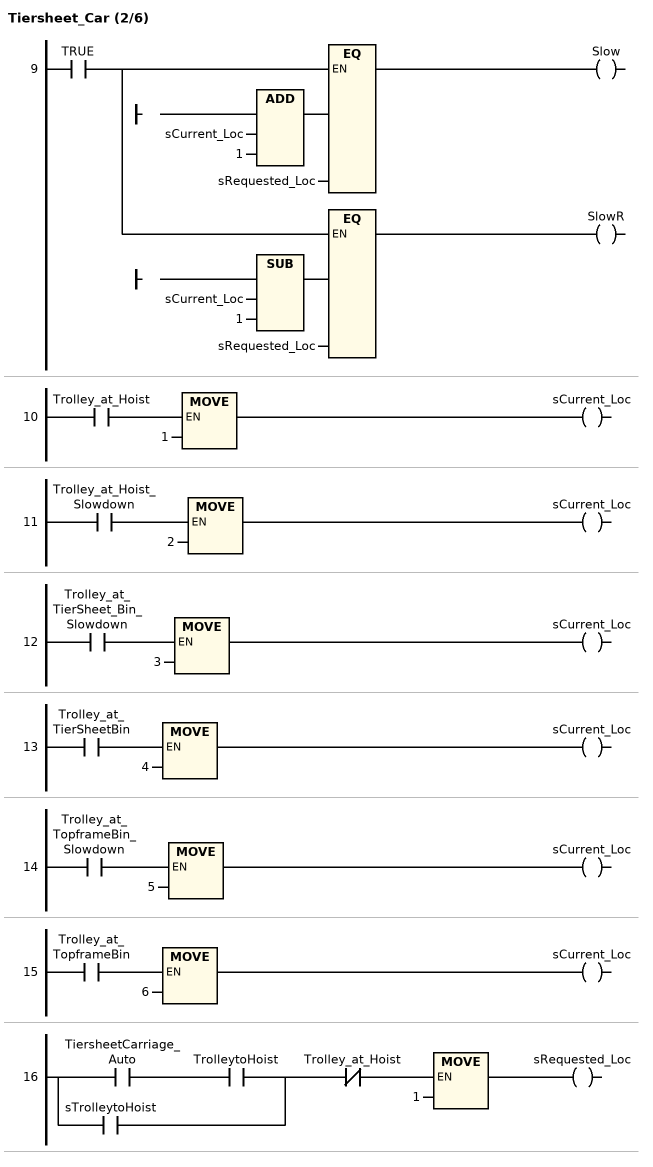
// NETWORK 9
Slow := sCurrent_Loc + 1 = sRequested_Loc;
SlowR := sCurrent_Loc - 1 = sRequested_Loc;

// NETWORK 10
IF Trolley_at_Hoist THEN _w1 := 1; END_IF
sCurrent_Loc := _w1;

// NETWORK 11
IF Trolley_at_Hoist_Slowdown THEN _w2 := 2; END_IF
sCurrent_Loc := _w2;

// NETWORK 12
IF Trolley_at_TierSheet_Bin_Slowdown THEN _w3 := 3; END_IF
sCurrent_Loc := _w3;

// NETWORK 13
IF Trolley_at_TierSheetBin THEN _w4 := 4; END_IF
sCurrent_Loc := _w4;

// NETWORK 14
IF Trolley_at_TopframeBin_Slowdown THEN _w5 := 5; END_IF
sCurrent_Loc := _w5;

// NETWORK 15
IF Trolley_at_TopframeBin THEN _w6 := 6; END_IF
sCurrent_Loc := _w6;

// NETWORK 16
IF (TiersheetCarriage_Auto AND TrolleytoHoist OR sTrolleytoHoist) AND NOT Trolley_at_Hoist THEN _w7 := 1; END_IF
sRequested_Loc := _w7;

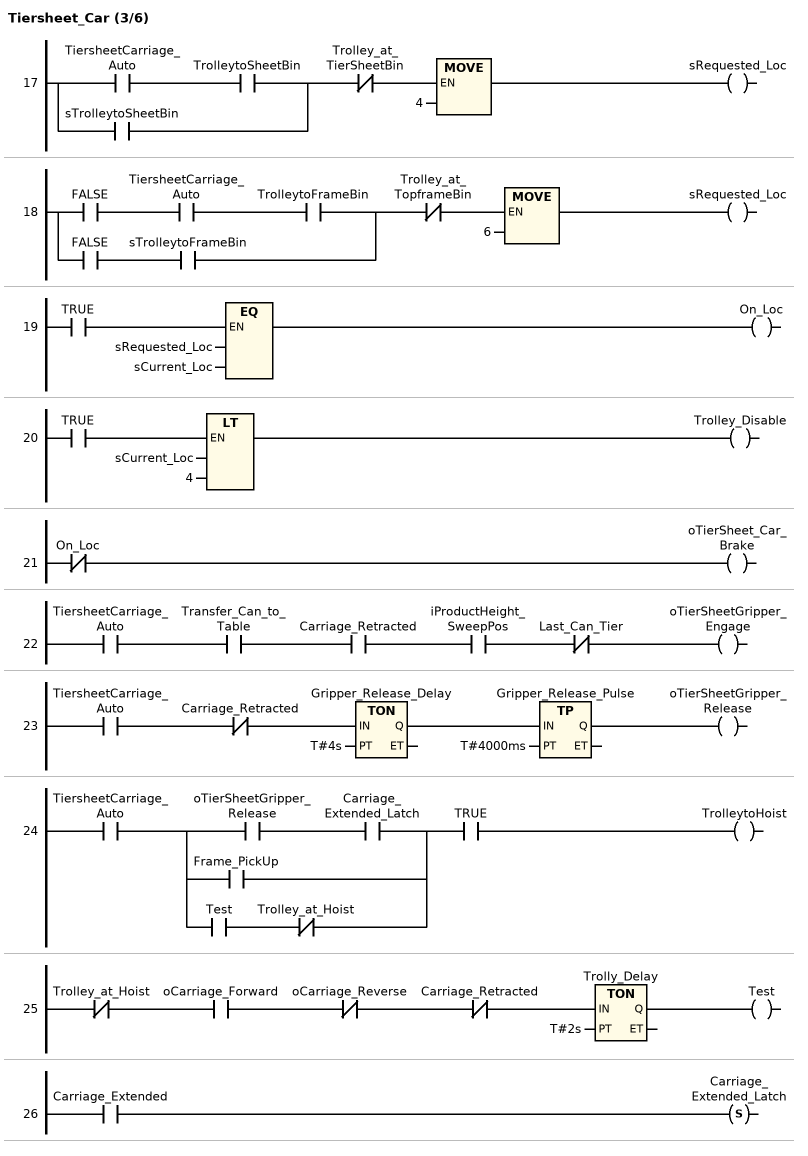
// NETWORK 17
IF (TiersheetCarriage_Auto AND TrolleytoSheetBin OR sTrolleytoSheetBin) AND NOT Trolley_at_TierSheetBin THEN
    _w8 := 4;
END_IF
sRequested_Loc := _w8;

// NETWORK 18
IF (FALSE AND TiersheetCarriage_Auto AND TrolleytoFrameBin OR FALSE AND sTrolleytoFrameBin) AND NOT Trolley_at_TopframeBin THEN
    _w9 := 6;
END_IF
sRequested_Loc := _w9;

// NETWORK 19
On_Loc := sRequested_Loc = sCurrent_Loc;

// NETWORK 20
Trolley_Disable := sCurrent_Loc < 4;

// NETWORK 21
oTierSheet_Car_Brake := NOT On_Loc;

// NETWORK 22
oTierSheetGripper_Engage := TiersheetCarriage_Auto AND Transfer_Can_to_Table AND Carriage_Retracted AND iProductHeight_SweepPos AND NOT Last_Can_Tier;

// NETWORK 23
Gripper_Release_Delay(IN := TiersheetCarriage_Auto AND NOT Carriage_Retracted, PT := T#4s); // TON
Gripper_Release_Pulse(IN := Gripper_Release_Delay.Q, PT := T#4000ms); // TP
oTierSheetGripper_Release := Gripper_Release_Pulse.Q;

// NETWORK 24
TrolleytoHoist := (TiersheetCarriage_Auto AND (oTierSheetGripper_Release AND Carriage_Extended_Latch OR Frame_PickUp OR Test AND NOT Trolley_at_Hoist)) AND TRUE;

// NETWORK 25
Trolly_Delay(IN := NOT Trolley_at_Hoist AND oCarriage_Forward AND NOT oCarriage_Reverse AND NOT Carriage_Retracted, PT := T#2s); // TON
Test := Trolly_Delay.Q;

// NETWORK 26
Carriage_Extended_Latch S= Carriage_Extended;

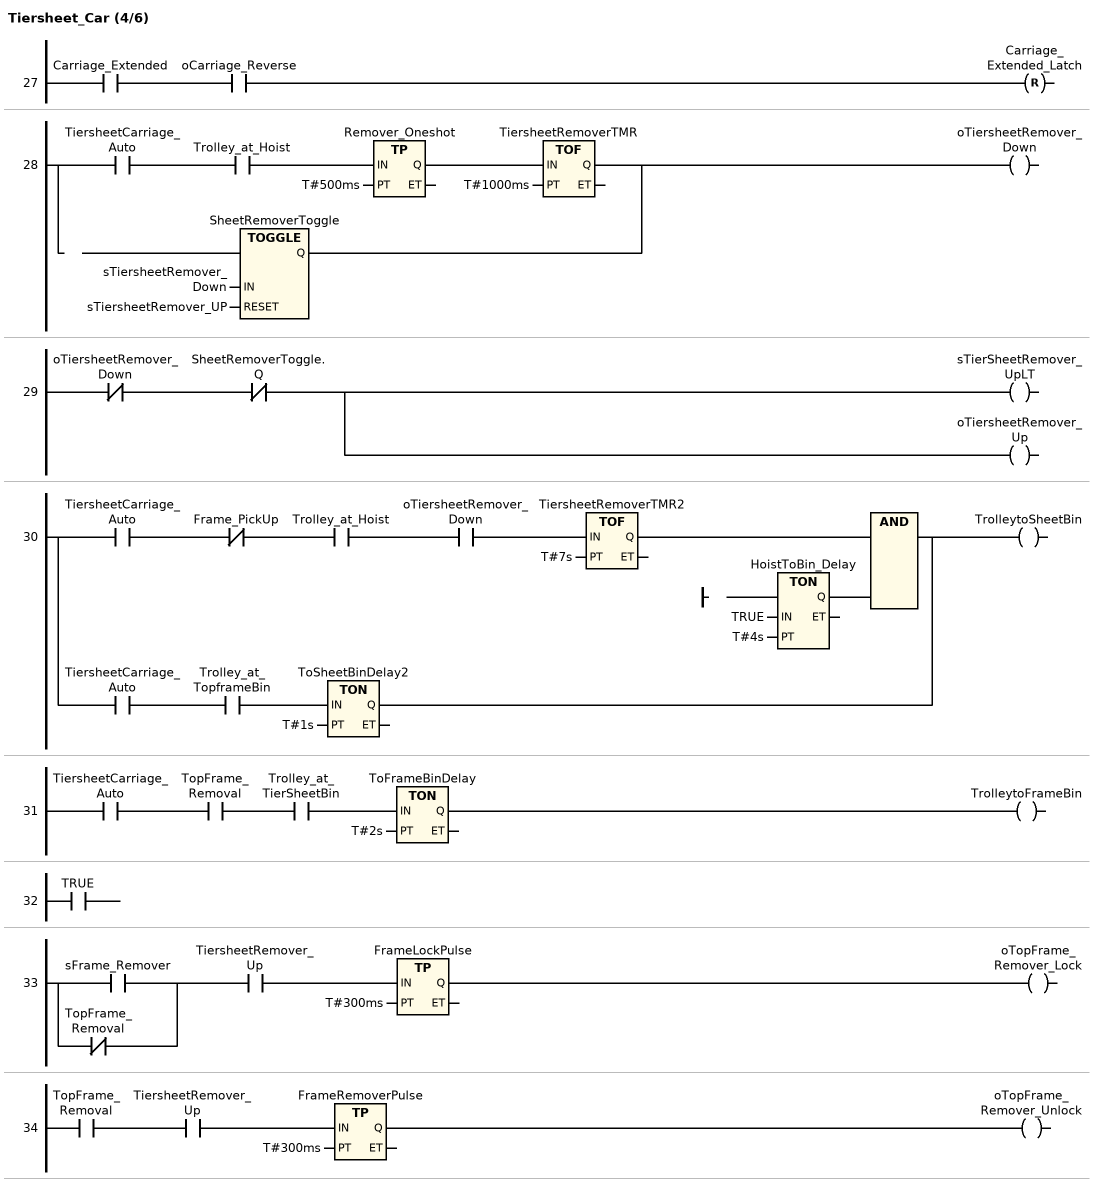
// NETWORK 27
Carriage_Extended_Latch R= Carriage_Extended AND oCarriage_Reverse;

// NETWORK 28
Remover_Oneshot(IN := TiersheetCarriage_Auto AND Trolley_at_Hoist, PT := T#500ms); // TP
TiersheetRemoverTMR(IN := Remover_Oneshot.Q, PT := T#1000ms); // TOF
SheetRemoverToggle(IN := sTiersheetRemover_Down, RESET := sTiersheetRemover_UP); // TOGGLE
oTiersheetRemover_Down := TiersheetRemoverTMR.Q OR SheetRemoverToggle.Q;

// NETWORK 29
_w10 := NOT oTiersheetRemover_Down AND NOT SheetRemoverToggle.Q;
sTierSheetRemover_UpLT := _w10;
oTiersheetRemover_Up := _w10;

// NETWORK 30
TiersheetRemoverTMR2(IN := TiersheetCarriage_Auto AND (NOT Frame_PickUp AND Trolley_at_Hoist AND oTiersheetRemover_Down), PT := T#7s); // TOF
HoistToBin_Delay(IN := TRUE, PT := T#4s); // TON
ToSheetBinDelay2(IN := TiersheetCarriage_Auto AND Trolley_at_TopframeBin, PT := T#1s); // TON
TrolleytoSheetBin := TiersheetRemoverTMR2.Q AND HoistToBin_Delay.Q OR ToSheetBinDelay2.Q;

// NETWORK 31
ToFrameBinDelay(IN := TiersheetCarriage_Auto AND TopFrame_Removal AND Trolley_at_TierSheetBin, PT := T#2s); // TON
TrolleytoFrameBin := ToFrameBinDelay.Q;

// NETWORK 32

// NETWORK 33
FrameLockPulse(IN := (sFrame_Remover OR NOT TopFrame_Removal) AND TiersheetRemover_Up, PT := T#300ms); // TP
oTopFrame_Remover_Lock := FrameLockPulse.Q;

// NETWORK 34
FrameRemoverPulse(IN := TopFrame_Removal AND TiersheetRemover_Up, PT := T#300ms); // TP
oTopFrame_Remover_Unlock := FrameRemoverPulse.Q;

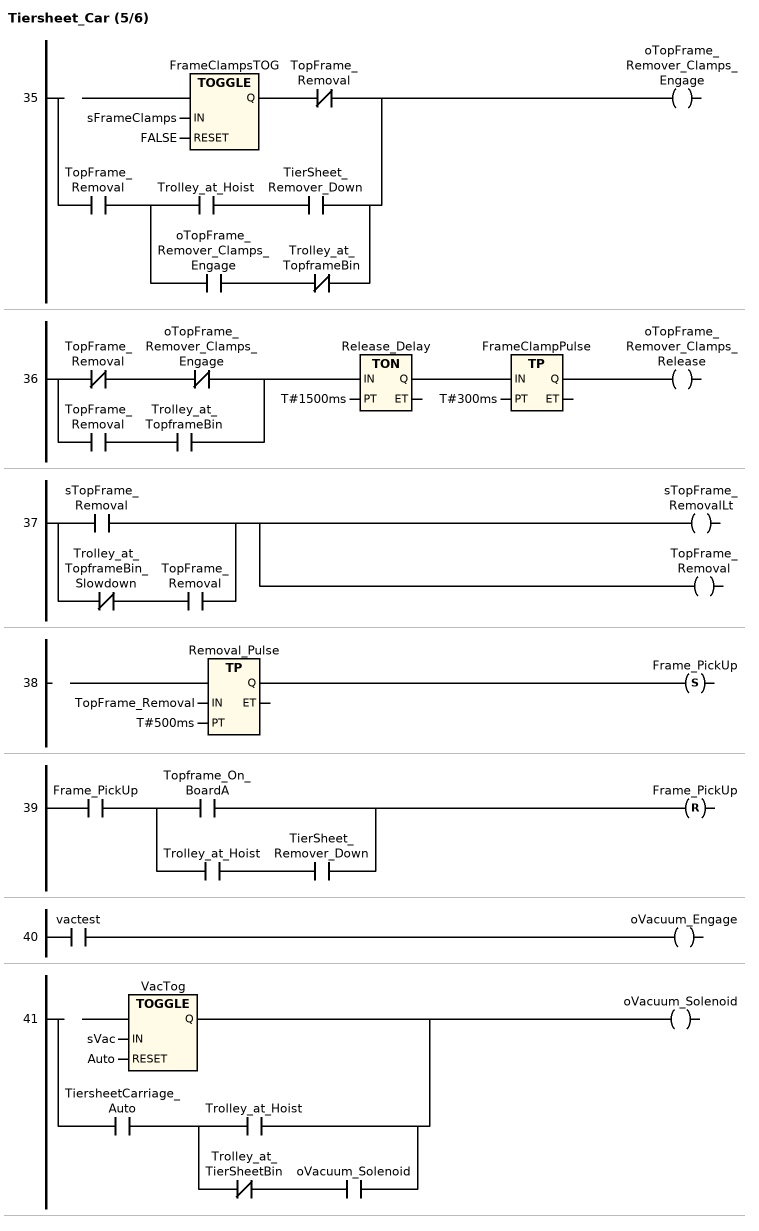
// NETWORK 35
FrameClampsTOG(IN := sFrameClamps, RESET := FALSE); // TOGGLE
oTopFrame_Remover_Clamps_Engage := FrameClampsTOG.Q AND NOT TopFrame_Removal OR TopFrame_Removal AND (Trolley_at_Hoist AND TierSheet_Remover_Down OR oTopFrame_Remover_Clamps_Engage AND NOT Trolley_at_TopframeBin);

// NETWORK 36
Release_Delay(IN := NOT TopFrame_Removal AND NOT oTopFrame_Remover_Clamps_Engage OR TopFrame_Removal AND Trolley_at_TopframeBin, PT := T#1500ms); // TON
FrameClampPulse(IN := Release_Delay.Q, PT := T#300ms); // TP
oTopFrame_Remover_Clamps_Release := FrameClampPulse.Q;

// NETWORK 37
_w11 := sTopFrame_Removal OR NOT Trolley_at_TopframeBin_Slowdown AND TopFrame_Removal;
sTopFrame_RemovalLt := _w11;
TopFrame_Removal := _w11;

// NETWORK 38
Removal_Pulse(IN := TopFrame_Removal, PT := T#500ms); // TP
Frame_PickUp S= Removal_Pulse.Q;

// NETWORK 39
Frame_PickUp R= Frame_PickUp AND (Topframe_On_BoardA OR Trolley_at_Hoist AND TierSheet_Remover_Down);

// NETWORK 40
oVacuum_Engage := vactest;

// NETWORK 41
VacTog(IN := sVac, RESET := Auto); // TOGGLE
oVacuum_Solenoid := VacTog.Q OR TiersheetCarriage_Auto AND (Trolley_at_Hoist OR NOT Trolley_at_TierSheetBin AND oVacuum_Solenoid);

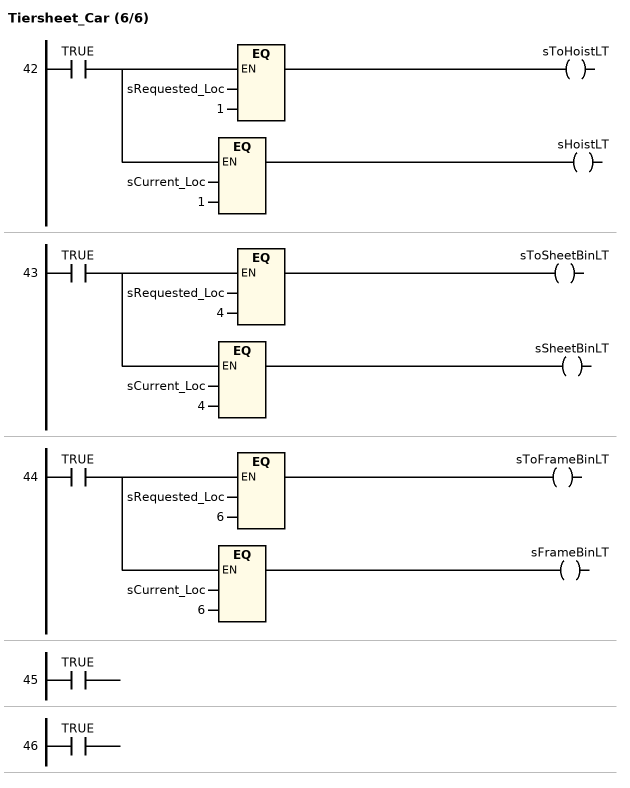
// NETWORK 42
sToHoistLT := sRequested_Loc = 1;
sHoistLT := sCurrent_Loc = 1;

// NETWORK 43
sToSheetBinLT := sRequested_Loc = 4;
sSheetBinLT := sCurrent_Loc = 4;

// NETWORK 44
sToFrameBinLT := sRequested_Loc = 6;
sFrameBinLT := sCurrent_Loc = 6;

// NETWORK 45

// NETWORK 46

END_PROGRAM

// ---- POUs/Messages.TcPOU
PROGRAM Messages
VAR

END_VAR

sMessages:='System Ok';


IF EmergencyStop_Latch THEN
	sMessages:='EMERGENCY  STOP!';
END_IF

END_PROGRAM
